// TIA Portal V17 export
// export: Created 2023-02-13T11:16:23.1750279Z, ExportSetting WithDefaults, DisplayName Totally Integrated Automation Portal, DisplayVersion V17, DisplayName TIA Portal Openness, DisplayVersion V17, DisplayName TIA Portal Teamcenter Gateway, DisplayVersion V17, DisplayName TIA Portal Version Control Interface, DisplayVersion V17, DisplayName SINAMICS Startdrive Advanced, DisplayVersion V17, DisplayName SINAMICS Startdrive G130, G150, S120, S150, SINAMICS MV, S210, DisplayVersion V17, DisplayName SINAMICS Startdrive G110M, G120, G120C, G120D, G120P, G115D, DisplayVersion V17, DisplayName STEP 7 Professional, DisplayVersion V17, DisplayName STEP 7 Safety, DisplayVersion V17, DisplayName WinCC Professional, DisplayVersion V17
FUNCTION_BLOCK "IO_Valve_Storage"   // FB1, LAD
{ S7_Optimized_Access := 'FALSE' }
VERSION : 0.1
// stored: AutoNumber true, IsIECCheckEnabled false, SetENOAutomatically false, UDAEnableTagReadback false
   VAR_INPUT
      lock : Bool;
      Init : Bool;
      Reset : Bool;
   END_VAR
   VAR
      "AV-23.01" { S7_SetPoint := 'True'} : "Valve";   // AUTO BUTTERFLY VALVE MAIN INLET PRODUCT TO STORAGE TANK T-23.00
      "AV-23.02" { S7_SetPoint := 'True'} : "Valve";   // AUTO BUTTERFLY VALVE CIP SUPPLY TO STORAGE TANK T-23.00 VIA PIPE INLET
      "AV-23.03" { S7_SetPoint := 'True'} : "Valve";   // AUTO BUTTERFLY VALVE INLET PRODUCT TO STORAGE TANK T-23.00
      "AV-23.04" { S7_SetPoint := 'True'} : "Valve";   // AUTO BUTTERFLY VALVE INLET PRODUCT FROM JBT TO STORAGE TANKS
      "AV-23.05" { S7_SetPoint := 'True'} : "Valve";   // AUTO BUTTERFLY VALVE INLET CIP PRODUCT FROM THE-4 TO STORAGE
      "AV-23.06" { S7_SetPoint := 'True'} : "Valve";   // AUTO BUTTERFLY VALVE OUTLET PRODUCT FROM STORAGE TANK T-23.00
      "AV-23.07" { S7_SetPoint := 'True'} : "Valve";   // AUTO BUTTERFLY VALVE CIP SUPPLY LINE STORAGE TANK T-23.00
      "AV-23.08" { S7_SetPoint := 'True'} : "Valve";   // AUTO BUTTERFLY VALVE CIP SUPPLY STORAGE TANK T-23.00 VIA SPRAY BALL
      "AV-24.01" { S7_SetPoint := 'True'} : "Valve";   // AUTO BUTTERFLY VALVE MAIN INLET PRODUCT TO STORAGE TANK T-24.00
      "AV-24.02" { S7_SetPoint := 'True'} : "Valve";   // AUTO BUTTERFLY VALVE CIP SUPPLY TO STORAGE TANK T-24.00 VIA PIPE INLET
      "AV-24.03" { S7_SetPoint := 'True'} : "Valve";   // AUTO BUTTERFLY VALVE INLET PRODUCT TO STORAGE TANK T-24.00
      "AV-24.04" { S7_SetPoint := 'True'} : "Valve";   // AUTO BUTTERFLY VALVE OUTLET PRODUCT FROM STORAGE TANK T-24.00
      "AV-24.05" { S7_SetPoint := 'True'} : "Valve";   // AUTO BUTTERFLY VALVE CIP SUPPLY LINE STORAGE TANK T-24.00
      "AV-24.06" { S7_SetPoint := 'True'} : "Valve";   // AUTO BUTTERFLY VALVE CIP SUPPLY STORAGE TANK T-24.00 VIA SPRAY BALL
      "AV-24.13" { S7_SetPoint := 'True'} : "Valve";   // AUTO BUTTERFLY VALVE MAIN INLET PRODUCT TO STORAGE TANK T-25.00
      "AV-24.14" { S7_SetPoint := 'True'} : "Valve";   // AUTO BUTTERFLY VALVE CIP SUPPLY TO STORAGE TANK T-25.00 VIA PIPE INLET
      "AV-29.01" { S7_SetPoint := 'True'} : "Valve";   // AUTO BUTTERFLY VALVE INLET PRODUCT TO STORAGE TANK T-25.00
      "AV-29.02" { S7_SetPoint := 'True'} : "Valve";   // AUTO BUTTERFLY VALVE OUTLET PRODUCT FROM STORAGE TANK T-25.00
      "AV-29.03" { S7_SetPoint := 'True'} : "Valve";   // AUTO BUTTERFLY VALVE CIP SUPPLY LINE STORAGE TANK T-25.00
      "AV-29.04" { S7_SetPoint := 'True'} : "Valve";   // AUTO BUTTERFLY VALVE CIP SUPPLY STORAGE TANK T-25.00 VIA SPRAY BALL
      "AV-29.06" { S7_SetPoint := 'True'} : "Valve";   // AUTO BUTTERFLY VALVE CIP SUPPLY STORAGE TANK T-25.00 VIA SPRAY BALL
      "AV-33.01" { S7_SetPoint := 'True'} : "Valve";   // AUTO BUTTERFLY VALVE CIP SUPPLY STORAGE TANKS FROM CIP SUPPLY LINE 3
      "AV-33.02" { S7_SetPoint := 'True'} : "Valve";   // AUTO BUTTERFLY VALVE CIP SUPPLY STORAGE TANK THE-4 JBT FROM CIP SUPPLY LINE 3
      "AV-33.03" { S7_SetPoint := 'True'} : "Valve";   // AUTO BUTTERFLY VALVE CIP SUPPLY STORAGE TANK THE-5 JBT FROM CIP SUPPLY LINE 3
      "AV-33.04" { S7_SetPoint := 'True'} : "Valve";   // AUTO BUTTERFLY VALVE MAIN CIP SUPPLY PRODUCT FROM THE-4 TO STORAGE
      "AV-33.05" { S7_SetPoint := 'True'} : "Valve";   // AUTO BUTTERFLY VALVE MAIN CIP SUPPLY TO STORAGE TANK T-23.00
      "AV-33.06" { S7_SetPoint := 'True'} : "Valve";   // AUTO BUTTERFLY VALVE MAIN CIP SUPPLY LINE STORAGE TANK T-23.00
      "AV-33.07" { S7_SetPoint := 'True'} : "Valve";   // AUTO BUTTERFLY VALVE MAIN CIP SUPPLY TO STORAGE TANK T-24.00
      "AV-33.08" { S7_SetPoint := 'True'} : "Valve";   // AUTO BUTTERFLY VALVE MAIN CIP SUPPLY LINE STORAGE TANK T-24.00
      "AV-33.09" { S7_SetPoint := 'True'} : "Valve";   // AUTO BUTTERFLY VALVE MAIN CIP SUPPLY TO STORAGE TANK T-25.00
      "AV-33.10" { S7_SetPoint := 'True'} : "Valve";
      "AV-33.11" { S7_SetPoint := 'True'} : "Valve";
      "AV-34.01" { S7_SetPoint := 'True'} : "Valve";
      "AV-34.02" { S7_SetPoint := 'True'} : "Valve";
      "AV-34.03" { S7_SetPoint := 'True'} : "Valve";
      "AV-34.04" { S7_SetPoint := 'True'} : "Valve";
      "AV-34.05" { S7_SetPoint := 'True'} : "Valve";
      "AV-34.06" { S7_SetPoint := 'True'} : "Valve";
      "AV-34.07" { S7_SetPoint := 'True'} : "Valve";
      "AV-34.08" { S7_SetPoint := 'True'} : "Valve";
      "AV-34.09" { S7_SetPoint := 'True'} : "Valve";
      "AV-34.10" { S7_SetPoint := 'True'} : "Valve";
      "AV-34.11" { S7_SetPoint := 'True'} : "Valve";
      "AV-34.12" { S7_SetPoint := 'True'} : "Valve";
      "AV-35.01" { S7_SetPoint := 'True'} : "Valve";
      "AV-35.02" { S7_SetPoint := 'True'} : "Valve";
      "AV-35.03" { S7_SetPoint := 'True'} : "Valve";
      "AV-35.04" { S7_SetPoint := 'True'} : "Valve";
      "AV-35.05" { S7_SetPoint := 'True'} : "Valve";
      "AV-35.06" { S7_SetPoint := 'True'} : "Valve";
      "AV-35.07" { S7_SetPoint := 'True'} : "Valve";
      "AV-35.08" { S7_SetPoint := 'True'} : "Valve";
      "AV-39.01" { S7_SetPoint := 'True'} : "Valve";
      "AV-39.02" { S7_SetPoint := 'True'} : "Valve";
      "AV-39.03" { S7_SetPoint := 'True'} : "Valve";
      "AV-39.04" { S7_SetPoint := 'True'} : "Valve";
      "AV-39.06" { S7_SetPoint := 'True'} : "Valve";
      "AV-24.15" { S7_SetPoint := 'True'} : "Valve";
      "AV-24.16" { S7_SetPoint := 'True'} : "Valve";
      "AV-79.01" { S7_SetPoint := 'True'} : "Valve";
      "AV-79.02" { S7_SetPoint := 'True'} : "Valve";
      "AV-79.03" { S7_SetPoint := 'True'} : "Valve";
      "AV-79.04" { S7_SetPoint := 'True'} : "Valve";
      "AV-79.05" { S7_SetPoint := 'True'} : "Valve";
      "AV-79.06" { S7_SetPoint := 'True'} : "Valve";
      "AV-79.07" { S7_SetPoint := 'True'} : "Valve";
      "AV-79.08" { S7_SetPoint := 'True'} : "Valve";
      "AV-79.09" { S7_SetPoint := 'True'} : "Valve";
      "AV-79.10" { S7_SetPoint := 'True'} : "Valve";
      "AV-79.13" { S7_SetPoint := 'True'} : "Valve";
      "AV-79.14" { S7_SetPoint := 'True'} : "Valve";
      "AV-79.15" { S7_SetPoint := 'True'} : "Valve";
      "AV-79.16" { S7_SetPoint := 'True'} : "Valve";
      "AV-79.17" { S7_SetPoint := 'True'} : "Valve";
      "AV-81.01" { S7_SetPoint := 'True'} : "Valve";
      "AV-81.02" { S7_SetPoint := 'True'} : "Valve";
      "AV-81.03" { S7_SetPoint := 'True'} : "Valve";
      "AV-81.04" { S7_SetPoint := 'True'} : "Valve";
      "AV-81.05" { S7_SetPoint := 'True'} : "Valve";
      "AV-81.06" { S7_SetPoint := 'True'} : "Valve";
      "AV-81.07" { S7_SetPoint := 'True'} : "Valve";
      "AV-81.08" { S7_SetPoint := 'True'} : "Valve";
      "AV-81.09" { S7_SetPoint := 'True'} : "Valve";
      "AV-81.10" { S7_SetPoint := 'True'} : "Valve";
      "AV-81.12" { S7_SetPoint := 'True'} : "Valve";
      "AV-81.13" { S7_SetPoint := 'True'} : "Valve";
      "AV-81.14" { S7_SetPoint := 'True'} : "Valve";
      "AV-85.01" { S7_SetPoint := 'True'} : "Valve";
      "AV-85.02" { S7_SetPoint := 'True'} : "Valve";
      "AV-85.03" { S7_SetPoint := 'True'} : "Valve";
      "AV-85.04" { S7_SetPoint := 'True'} : "Valve";
      "AV-85.13" { S7_SetPoint := 'True'} : "Valve";
      "AV-85.12" { S7_SetPoint := 'True'} : "Valve";
      "AV-85.14" { S7_SetPoint := 'True'} : "Valve";
      "AV-85.15" { S7_SetPoint := 'True'} : "Valve";
      "AV-85.05" { S7_SetPoint := 'True'} : "Valve";
      "AV-85.06" { S7_SetPoint := 'True'} : "Valve";
      "AV-85.16" { S7_SetPoint := 'True'} : "Valve";
      "AV-85.17" { S7_SetPoint := 'True'} : "Valve";
      "AV-85.18" { S7_SetPoint := 'True'} : "Valve";
      "AV-85.09" { S7_SetPoint := 'True'} : "Valve";
      "AV-85.08" { S7_SetPoint := 'True'} : "Valve";
      "AV-85.10" { S7_SetPoint := 'True'} : "Valve";
      "AV-85.11" { S7_SetPoint := 'True'} : "Valve";
      "AV-84.05" { S7_SetPoint := 'True'} : "Valve";
      "AV-84.06" { S7_SetPoint := 'True'} : "Valve";
      "AV-84.07" { S7_SetPoint := 'True'} : "Valve";
      "AV-84.08" { S7_SetPoint := 'True'} : "Valve";
      "AV-84.09" { S7_SetPoint := 'True'} : "Valve";
      "AV-84.10" { S7_SetPoint := 'True'} : "Valve";
      "AV-84.12" { S7_SetPoint := 'True'} : "Valve";
      "AV-84.13" { S7_SetPoint := 'True'} : "Valve";
      "AV-84.14" { S7_SetPoint := 'True'} : "Valve";
      "AV-24.09" { S7_SetPoint := 'True'} : "Valve";
      "AV-24.17" { S7_SetPoint := 'True'} : "Valve";
      "AV-24.18" { S7_SetPoint := 'True'} : "Valve";
      "AV-24.19" { S7_SetPoint := 'True'} : "Valve";
      "AV-24.20" { S7_SetPoint := 'True'} : "Valve";
      "AV-24.21" { S7_SetPoint := 'True'} : "Valve";
      "AV-24.22" { S7_SetPoint := 'True'} : "Valve";
      "AV-24.23" { S7_SetPoint := 'True'} : "Valve";
      "AV-24.24" { S7_SetPoint := 'True'} : "Valve";
      "AV-79.21" { S7_SetPoint := 'True'} : "Valve";
      "AV-79.18" { S7_SetPoint := 'True'} : "Valve";
      "AV-79.19" { S7_SetPoint := 'True'} : "Valve";
      "AV-79.20" { S7_SetPoint := 'True'} : "Valve";
   END_VAR
BEGIN

REGION Network 1: AV-23.01
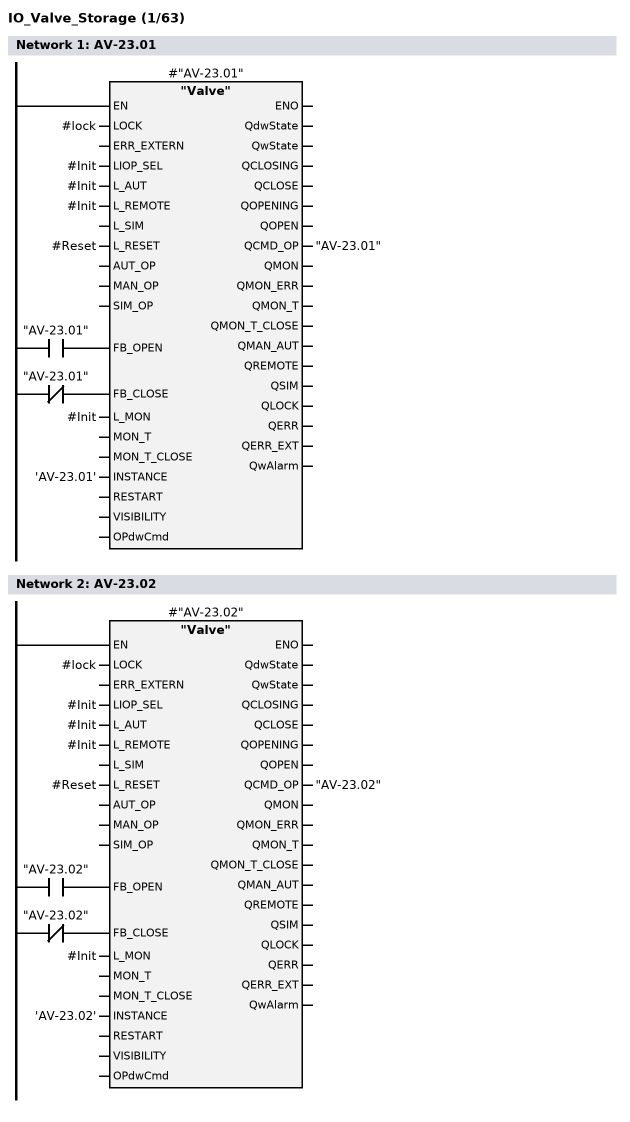
   RUNG wire#powerrail
      #"AV-23.01"(FB_OPEN := wire#w1, FB_CLOSE := wire#w2, LOCK := #lock, ERR_EXTERN :=, LIOP_SEL := #Init, L_AUT := #Init, L_REMOTE := #Init, L_SIM :=, L_RESET := #Reset, AUT_OP :=, MAN_OP :=, SIM_OP :=, L_MON := #Init, MON_T :=, MON_T_CLOSE :=, INSTANCE := 'AV-23.01', RESTART :=, VISIBILITY :=, OPdwCmd :=, QdwState =>, QwState =>, QCLOSING =>, QCLOSE =>, QOPENING =>, QOPEN =>, QCMD_OP => "AV-23.01", QMON =>, QMON_ERR =>, QMON_T =>, QMON_T_CLOSE =>, QMAN_AUT =>, QREMOTE =>, QSIM =>, QLOCK =>, QERR =>, QERR_EXT =>, QwAlarm =>)
   END_RUNG
   RUNG wire#powerrail
      Contact( "AV-23.01" )
   END_RUNG wire#w1
   RUNG wire#powerrail
      I_Contact( "AV-23.01" )
   END_RUNG wire#w2
   // the same network as SCL:
   #"AV-23.01"(LOCK := #lock,   // "Valve"
               LIOP_SEL := #Init,
               L_AUT := #Init,
               L_REMOTE := #Init,
               L_RESET := #Reset,
               FB_OPEN := "AV-23.01",
               FB_CLOSE := NOT "AV-23.01",
               L_MON := #Init,
               INSTANCE := 'AV-23.01',
               QCMD_OP => "AV-23.01");
END_REGION

REGION Network 2: AV-23.02
   RUNG wire#powerrail
      #"AV-23.02"(FB_OPEN := wire#w1, FB_CLOSE := wire#w2, LOCK := #lock, ERR_EXTERN :=, LIOP_SEL := #Init, L_AUT := #Init, L_REMOTE := #Init, L_SIM :=, L_RESET := #Reset, AUT_OP :=, MAN_OP :=, SIM_OP :=, L_MON := #Init, MON_T :=, MON_T_CLOSE :=, INSTANCE := 'AV-23.02', RESTART :=, VISIBILITY :=, OPdwCmd :=, QdwState =>, QwState =>, QCLOSING =>, QCLOSE =>, QOPENING =>, QOPEN =>, QCMD_OP => "AV-23.02", QMON =>, QMON_ERR =>, QMON_T =>, QMON_T_CLOSE =>, QMAN_AUT =>, QREMOTE =>, QSIM =>, QLOCK =>, QERR =>, QERR_EXT =>, QwAlarm =>)
   END_RUNG
   RUNG wire#powerrail
      Contact( "AV-23.02" )
   END_RUNG wire#w1
   RUNG wire#powerrail
      I_Contact( "AV-23.02" )
   END_RUNG wire#w2
   // the same network as SCL:
   #"AV-23.02"(LOCK := #lock,   // "Valve"
               LIOP_SEL := #Init,
               L_AUT := #Init,
               L_REMOTE := #Init,
               L_RESET := #Reset,
               FB_OPEN := "AV-23.02",
               FB_CLOSE := NOT "AV-23.02",
               L_MON := #Init,
               INSTANCE := 'AV-23.02',
               QCMD_OP => "AV-23.02");
END_REGION

REGION Network 3: AV-23.03
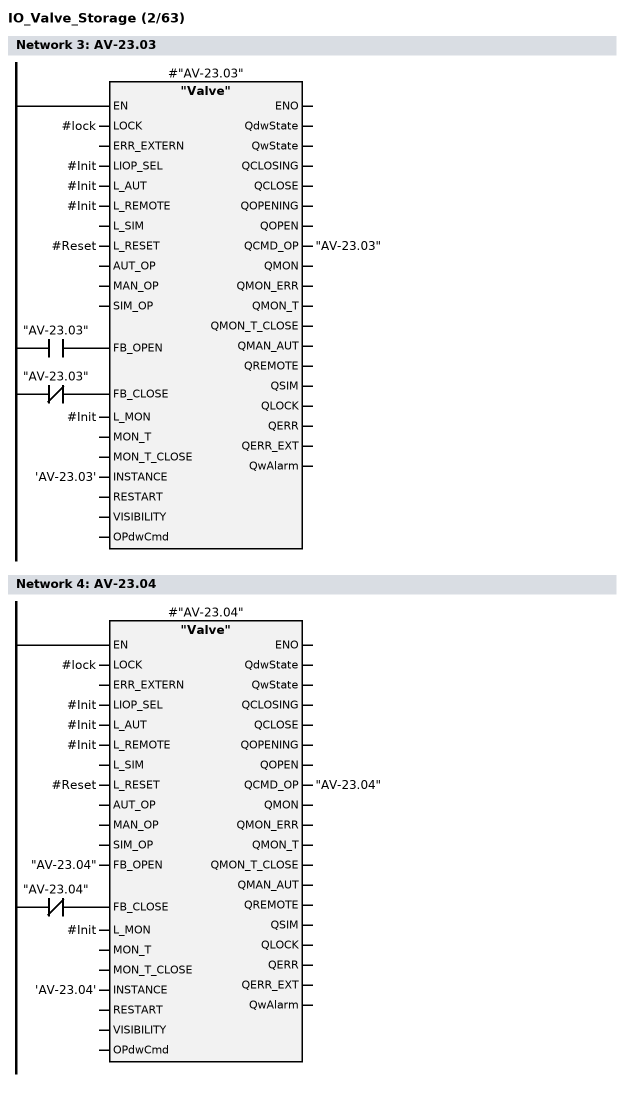
   RUNG wire#powerrail
      #"AV-23.03"(FB_OPEN := wire#w1, FB_CLOSE := wire#w2, LOCK := #lock, ERR_EXTERN :=, LIOP_SEL := #Init, L_AUT := #Init, L_REMOTE := #Init, L_SIM :=, L_RESET := #Reset, AUT_OP :=, MAN_OP :=, SIM_OP :=, L_MON := #Init, MON_T :=, MON_T_CLOSE :=, INSTANCE := 'AV-23.03', RESTART :=, VISIBILITY :=, OPdwCmd :=, QdwState =>, QwState =>, QCLOSING =>, QCLOSE =>, QOPENING =>, QOPEN =>, QCMD_OP => "AV-23.03", QMON =>, QMON_ERR =>, QMON_T =>, QMON_T_CLOSE =>, QMAN_AUT =>, QREMOTE =>, QSIM =>, QLOCK =>, QERR =>, QERR_EXT =>, QwAlarm =>)
   END_RUNG
   RUNG wire#powerrail
      Contact( "AV-23.03" )
   END_RUNG wire#w1
   RUNG wire#powerrail
      I_Contact( "AV-23.03" )
   END_RUNG wire#w2
   // the same network as SCL:
   #"AV-23.03"(LOCK := #lock,   // "Valve"
               LIOP_SEL := #Init,
               L_AUT := #Init,
               L_REMOTE := #Init,
               L_RESET := #Reset,
               FB_OPEN := "AV-23.03",
               FB_CLOSE := NOT "AV-23.03",
               L_MON := #Init,
               INSTANCE := 'AV-23.03',
               QCMD_OP => "AV-23.03");
END_REGION

REGION Network 4: AV-23.04
   RUNG wire#powerrail
      #"AV-23.04"(FB_CLOSE := wire#w1, LOCK := #lock, ERR_EXTERN :=, LIOP_SEL := #Init, L_AUT := #Init, L_REMOTE := #Init, L_SIM :=, L_RESET := #Reset, AUT_OP :=, MAN_OP :=, SIM_OP :=, FB_OPEN := "AV-23.04", L_MON := #Init, MON_T :=, MON_T_CLOSE :=, INSTANCE := 'AV-23.04', RESTART :=, VISIBILITY :=, OPdwCmd :=, QdwState =>, QwState =>, QCLOSING =>, QCLOSE =>, QOPENING =>, QOPEN =>, QCMD_OP => "AV-23.04", QMON =>, QMON_ERR =>, QMON_T =>, QMON_T_CLOSE =>, QMAN_AUT =>, QREMOTE =>, QSIM =>, QLOCK =>, QERR =>, QERR_EXT =>, QwAlarm =>)
   END_RUNG
   RUNG wire#powerrail
      I_Contact( "AV-23.04" )
   END_RUNG wire#w1
   // the same network as SCL:
   #"AV-23.04"(LOCK := #lock,   // "Valve"
               LIOP_SEL := #Init,
               L_AUT := #Init,
               L_REMOTE := #Init,
               L_RESET := #Reset,
               FB_OPEN := "AV-23.04",
               FB_CLOSE := NOT "AV-23.04",
               L_MON := #Init,
               INSTANCE := 'AV-23.04',
               QCMD_OP => "AV-23.04");
END_REGION

REGION Network 5: AV-23.05
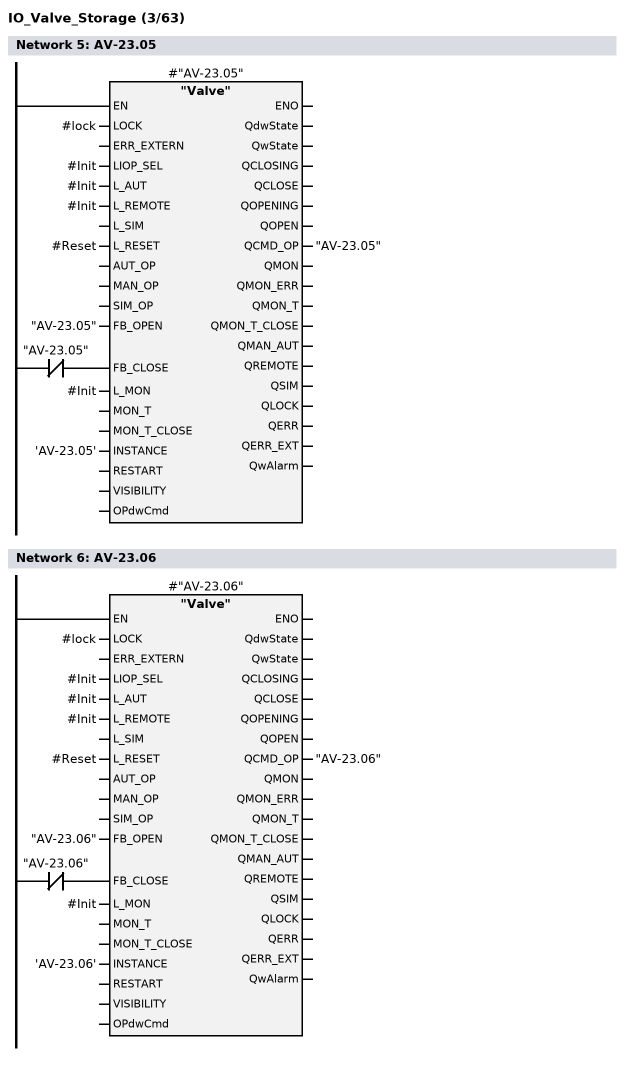
   RUNG wire#powerrail
      #"AV-23.05"(FB_CLOSE := wire#w1, LOCK := #lock, ERR_EXTERN :=, LIOP_SEL := #Init, L_AUT := #Init, L_REMOTE := #Init, L_SIM :=, L_RESET := #Reset, AUT_OP :=, MAN_OP :=, SIM_OP :=, FB_OPEN := "AV-23.05", L_MON := #Init, MON_T :=, MON_T_CLOSE :=, INSTANCE := 'AV-23.05', RESTART :=, VISIBILITY :=, OPdwCmd :=, QdwState =>, QwState =>, QCLOSING =>, QCLOSE =>, QOPENING =>, QOPEN =>, QCMD_OP => "AV-23.05", QMON =>, QMON_ERR =>, QMON_T =>, QMON_T_CLOSE =>, QMAN_AUT =>, QREMOTE =>, QSIM =>, QLOCK =>, QERR =>, QERR_EXT =>, QwAlarm =>)
   END_RUNG
   RUNG wire#powerrail
      I_Contact( "AV-23.05" )
   END_RUNG wire#w1
   // the same network as SCL:
   #"AV-23.05"(LOCK := #lock,   // "Valve"
               LIOP_SEL := #Init,
               L_AUT := #Init,
               L_REMOTE := #Init,
               L_RESET := #Reset,
               FB_OPEN := "AV-23.05",
               FB_CLOSE := NOT "AV-23.05",
               L_MON := #Init,
               INSTANCE := 'AV-23.05',
               QCMD_OP => "AV-23.05");
END_REGION

REGION Network 6: AV-23.06
   RUNG wire#powerrail
      #"AV-23.06"(FB_CLOSE := wire#w1, LOCK := #lock, ERR_EXTERN :=, LIOP_SEL := #Init, L_AUT := #Init, L_REMOTE := #Init, L_SIM :=, L_RESET := #Reset, AUT_OP :=, MAN_OP :=, SIM_OP :=, FB_OPEN := "AV-23.06", L_MON := #Init, MON_T :=, MON_T_CLOSE :=, INSTANCE := 'AV-23.06', RESTART :=, VISIBILITY :=, OPdwCmd :=, QdwState =>, QwState =>, QCLOSING =>, QCLOSE =>, QOPENING =>, QOPEN =>, QCMD_OP => "AV-23.06", QMON =>, QMON_ERR =>, QMON_T =>, QMON_T_CLOSE =>, QMAN_AUT =>, QREMOTE =>, QSIM =>, QLOCK =>, QERR =>, QERR_EXT =>, QwAlarm =>)
   END_RUNG
   RUNG wire#powerrail
      I_Contact( "AV-23.06" )
   END_RUNG wire#w1
   // the same network as SCL:
   #"AV-23.06"(LOCK := #lock,   // "Valve"
               LIOP_SEL := #Init,
               L_AUT := #Init,
               L_REMOTE := #Init,
               L_RESET := #Reset,
               FB_OPEN := "AV-23.06",
               FB_CLOSE := NOT "AV-23.06",
               L_MON := #Init,
               INSTANCE := 'AV-23.06',
               QCMD_OP => "AV-23.06");
END_REGION

REGION Network 7: AV-23.07
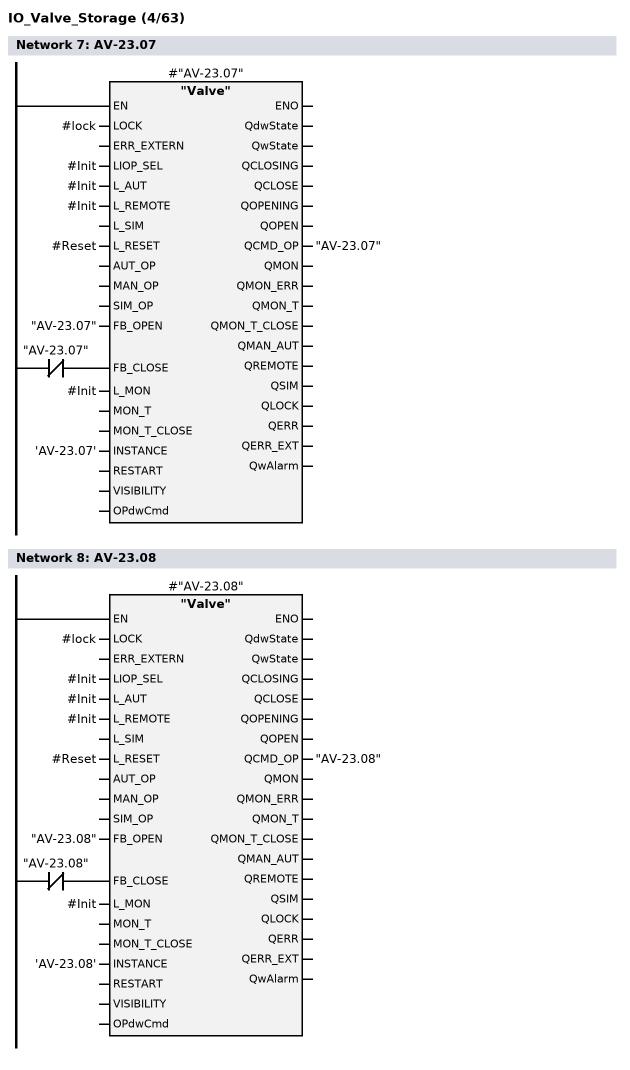
   RUNG wire#powerrail
      #"AV-23.07"(FB_CLOSE := wire#w1, LOCK := #lock, ERR_EXTERN :=, LIOP_SEL := #Init, L_AUT := #Init, L_REMOTE := #Init, L_SIM :=, L_RESET := #Reset, AUT_OP :=, MAN_OP :=, SIM_OP :=, FB_OPEN := "AV-23.07", L_MON := #Init, MON_T :=, MON_T_CLOSE :=, INSTANCE := 'AV-23.07', RESTART :=, VISIBILITY :=, OPdwCmd :=, QdwState =>, QwState =>, QCLOSING =>, QCLOSE =>, QOPENING =>, QOPEN =>, QCMD_OP => "AV-23.07", QMON =>, QMON_ERR =>, QMON_T =>, QMON_T_CLOSE =>, QMAN_AUT =>, QREMOTE =>, QSIM =>, QLOCK =>, QERR =>, QERR_EXT =>, QwAlarm =>)
   END_RUNG
   RUNG wire#powerrail
      I_Contact( "AV-23.07" )
   END_RUNG wire#w1
   // the same network as SCL:
   #"AV-23.07"(LOCK := #lock,   // "Valve"
               LIOP_SEL := #Init,
               L_AUT := #Init,
               L_REMOTE := #Init,
               L_RESET := #Reset,
               FB_OPEN := "AV-23.07",
               FB_CLOSE := NOT "AV-23.07",
               L_MON := #Init,
               INSTANCE := 'AV-23.07',
               QCMD_OP => "AV-23.07");
END_REGION

REGION Network 8: AV-23.08
   RUNG wire#powerrail
      #"AV-23.08"(FB_CLOSE := wire#w1, LOCK := #lock, ERR_EXTERN :=, LIOP_SEL := #Init, L_AUT := #Init, L_REMOTE := #Init, L_SIM :=, L_RESET := #Reset, AUT_OP :=, MAN_OP :=, SIM_OP :=, FB_OPEN := "AV-23.08", L_MON := #Init, MON_T :=, MON_T_CLOSE :=, INSTANCE := 'AV-23.08', RESTART :=, VISIBILITY :=, OPdwCmd :=, QdwState =>, QwState =>, QCLOSING =>, QCLOSE =>, QOPENING =>, QOPEN =>, QCMD_OP => "AV-23.08", QMON =>, QMON_ERR =>, QMON_T =>, QMON_T_CLOSE =>, QMAN_AUT =>, QREMOTE =>, QSIM =>, QLOCK =>, QERR =>, QERR_EXT =>, QwAlarm =>)
   END_RUNG
   RUNG wire#powerrail
      I_Contact( "AV-23.08" )
   END_RUNG wire#w1
   // the same network as SCL:
   #"AV-23.08"(LOCK := #lock,   // "Valve"
               LIOP_SEL := #Init,
               L_AUT := #Init,
               L_REMOTE := #Init,
               L_RESET := #Reset,
               FB_OPEN := "AV-23.08",
               FB_CLOSE := NOT "AV-23.08",
               L_MON := #Init,
               INSTANCE := 'AV-23.08',
               QCMD_OP => "AV-23.08");
END_REGION

REGION Network 10: AV-24.01
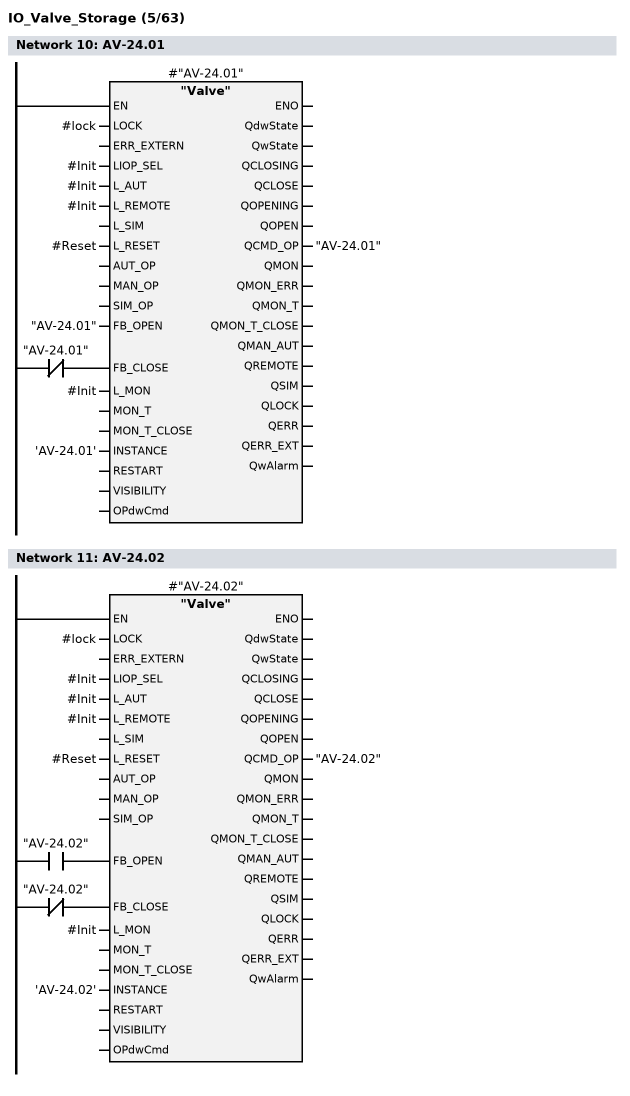
   RUNG wire#powerrail
      #"AV-24.01"(FB_CLOSE := wire#w1, LOCK := #lock, ERR_EXTERN :=, LIOP_SEL := #Init, L_AUT := #Init, L_REMOTE := #Init, L_SIM :=, L_RESET := #Reset, AUT_OP :=, MAN_OP :=, SIM_OP :=, FB_OPEN := "AV-24.01", L_MON := #Init, MON_T :=, MON_T_CLOSE :=, INSTANCE := 'AV-24.01', RESTART :=, VISIBILITY :=, OPdwCmd :=, QdwState =>, QwState =>, QCLOSING =>, QCLOSE =>, QOPENING =>, QOPEN =>, QCMD_OP => "AV-24.01", QMON =>, QMON_ERR =>, QMON_T =>, QMON_T_CLOSE =>, QMAN_AUT =>, QREMOTE =>, QSIM =>, QLOCK =>, QERR =>, QERR_EXT =>, QwAlarm =>)
   END_RUNG
   RUNG wire#powerrail
      I_Contact( "AV-24.01" )
   END_RUNG wire#w1
   // the same network as SCL:
   #"AV-24.01"(LOCK := #lock,   // "Valve"
               LIOP_SEL := #Init,
               L_AUT := #Init,
               L_REMOTE := #Init,
               L_RESET := #Reset,
               FB_OPEN := "AV-24.01",
               FB_CLOSE := NOT "AV-24.01",
               L_MON := #Init,
               INSTANCE := 'AV-24.01',
               QCMD_OP => "AV-24.01");
END_REGION

REGION Network 11: AV-24.02
   RUNG wire#powerrail
      #"AV-24.02"(FB_OPEN := wire#w1, FB_CLOSE := wire#w2, LOCK := #lock, ERR_EXTERN :=, LIOP_SEL := #Init, L_AUT := #Init, L_REMOTE := #Init, L_SIM :=, L_RESET := #Reset, AUT_OP :=, MAN_OP :=, SIM_OP :=, L_MON := #Init, MON_T :=, MON_T_CLOSE :=, INSTANCE := 'AV-24.02', RESTART :=, VISIBILITY :=, OPdwCmd :=, QdwState =>, QwState =>, QCLOSING =>, QCLOSE =>, QOPENING =>, QOPEN =>, QCMD_OP => "AV-24.02", QMON =>, QMON_ERR =>, QMON_T =>, QMON_T_CLOSE =>, QMAN_AUT =>, QREMOTE =>, QSIM =>, QLOCK =>, QERR =>, QERR_EXT =>, QwAlarm =>)
   END_RUNG
   RUNG wire#powerrail
      Contact( "AV-24.02" )
   END_RUNG wire#w1
   RUNG wire#powerrail
      I_Contact( "AV-24.02" )
   END_RUNG wire#w2
   // the same network as SCL:
   #"AV-24.02"(LOCK := #lock,   // "Valve"
               LIOP_SEL := #Init,
               L_AUT := #Init,
               L_REMOTE := #Init,
               L_RESET := #Reset,
               FB_OPEN := "AV-24.02",
               FB_CLOSE := NOT "AV-24.02",
               L_MON := #Init,
               INSTANCE := 'AV-24.02',
               QCMD_OP => "AV-24.02");
END_REGION

REGION Network 12: AV-24.03
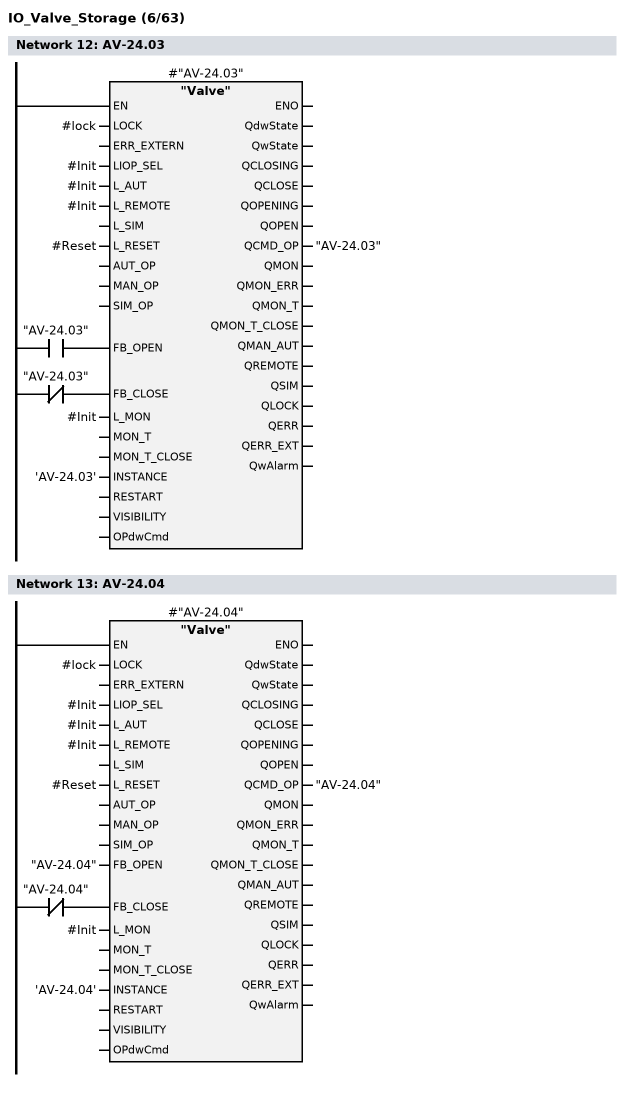
   RUNG wire#powerrail
      #"AV-24.03"(FB_OPEN := wire#w1, FB_CLOSE := wire#w2, LOCK := #lock, ERR_EXTERN :=, LIOP_SEL := #Init, L_AUT := #Init, L_REMOTE := #Init, L_SIM :=, L_RESET := #Reset, AUT_OP :=, MAN_OP :=, SIM_OP :=, L_MON := #Init, MON_T :=, MON_T_CLOSE :=, INSTANCE := 'AV-24.03', RESTART :=, VISIBILITY :=, OPdwCmd :=, QdwState =>, QwState =>, QCLOSING =>, QCLOSE =>, QOPENING =>, QOPEN =>, QCMD_OP => "AV-24.03", QMON =>, QMON_ERR =>, QMON_T =>, QMON_T_CLOSE =>, QMAN_AUT =>, QREMOTE =>, QSIM =>, QLOCK =>, QERR =>, QERR_EXT =>, QwAlarm =>)
   END_RUNG
   RUNG wire#powerrail
      Contact( "AV-24.03" )
   END_RUNG wire#w1
   RUNG wire#powerrail
      I_Contact( "AV-24.03" )
   END_RUNG wire#w2
   // the same network as SCL:
   #"AV-24.03"(LOCK := #lock,   // "Valve"
               LIOP_SEL := #Init,
               L_AUT := #Init,
               L_REMOTE := #Init,
               L_RESET := #Reset,
               FB_OPEN := "AV-24.03",
               FB_CLOSE := NOT "AV-24.03",
               L_MON := #Init,
               INSTANCE := 'AV-24.03',
               QCMD_OP => "AV-24.03");
END_REGION

REGION Network 13: AV-24.04
   RUNG wire#powerrail
      #"AV-24.04"(FB_CLOSE := wire#w1, LOCK := #lock, ERR_EXTERN :=, LIOP_SEL := #Init, L_AUT := #Init, L_REMOTE := #Init, L_SIM :=, L_RESET := #Reset, AUT_OP :=, MAN_OP :=, SIM_OP :=, FB_OPEN := "AV-24.04", L_MON := #Init, MON_T :=, MON_T_CLOSE :=, INSTANCE := 'AV-24.04', RESTART :=, VISIBILITY :=, OPdwCmd :=, QdwState =>, QwState =>, QCLOSING =>, QCLOSE =>, QOPENING =>, QOPEN =>, QCMD_OP => "AV-24.04", QMON =>, QMON_ERR =>, QMON_T =>, QMON_T_CLOSE =>, QMAN_AUT =>, QREMOTE =>, QSIM =>, QLOCK =>, QERR =>, QERR_EXT =>, QwAlarm =>)
   END_RUNG
   RUNG wire#powerrail
      I_Contact( "AV-24.04" )
   END_RUNG wire#w1
   // the same network as SCL:
   #"AV-24.04"(LOCK := #lock,   // "Valve"
               LIOP_SEL := #Init,
               L_AUT := #Init,
               L_REMOTE := #Init,
               L_RESET := #Reset,
               FB_OPEN := "AV-24.04",
               FB_CLOSE := NOT "AV-24.04",
               L_MON := #Init,
               INSTANCE := 'AV-24.04',
               QCMD_OP => "AV-24.04");
END_REGION

REGION Network 14: AV-24.05
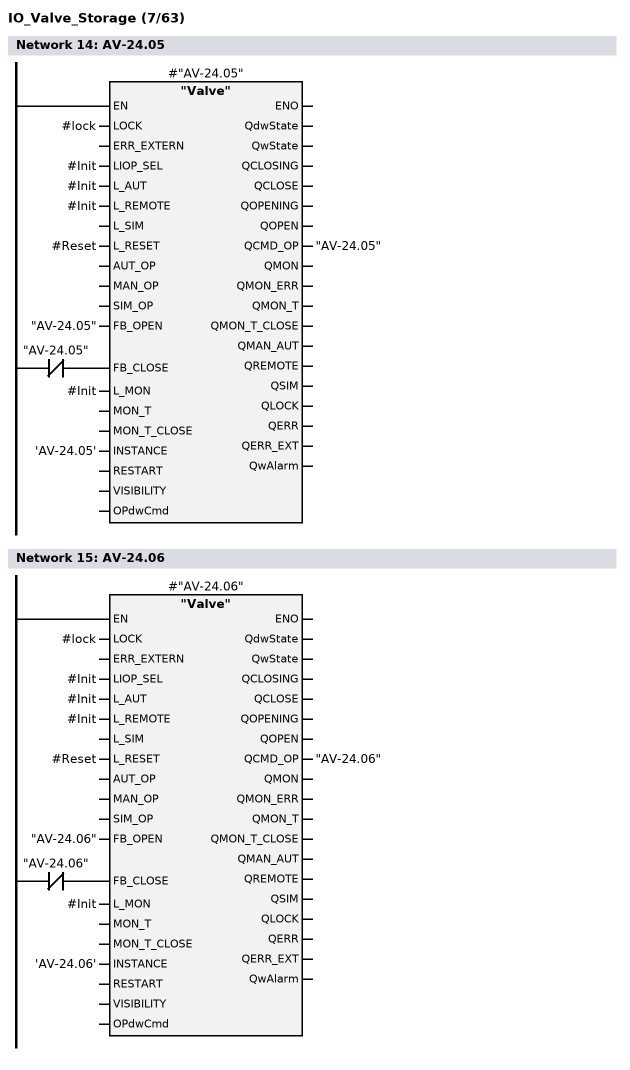
   RUNG wire#powerrail
      #"AV-24.05"(FB_CLOSE := wire#w1, LOCK := #lock, ERR_EXTERN :=, LIOP_SEL := #Init, L_AUT := #Init, L_REMOTE := #Init, L_SIM :=, L_RESET := #Reset, AUT_OP :=, MAN_OP :=, SIM_OP :=, FB_OPEN := "AV-24.05", L_MON := #Init, MON_T :=, MON_T_CLOSE :=, INSTANCE := 'AV-24.05', RESTART :=, VISIBILITY :=, OPdwCmd :=, QdwState =>, QwState =>, QCLOSING =>, QCLOSE =>, QOPENING =>, QOPEN =>, QCMD_OP => "AV-24.05", QMON =>, QMON_ERR =>, QMON_T =>, QMON_T_CLOSE =>, QMAN_AUT =>, QREMOTE =>, QSIM =>, QLOCK =>, QERR =>, QERR_EXT =>, QwAlarm =>)
   END_RUNG
   RUNG wire#powerrail
      I_Contact( "AV-24.05" )
   END_RUNG wire#w1
   // the same network as SCL:
   #"AV-24.05"(LOCK := #lock,   // "Valve"
               LIOP_SEL := #Init,
               L_AUT := #Init,
               L_REMOTE := #Init,
               L_RESET := #Reset,
               FB_OPEN := "AV-24.05",
               FB_CLOSE := NOT "AV-24.05",
               L_MON := #Init,
               INSTANCE := 'AV-24.05',
               QCMD_OP => "AV-24.05");
END_REGION

REGION Network 15: AV-24.06
   RUNG wire#powerrail
      #"AV-24.06"(FB_CLOSE := wire#w1, LOCK := #lock, ERR_EXTERN :=, LIOP_SEL := #Init, L_AUT := #Init, L_REMOTE := #Init, L_SIM :=, L_RESET := #Reset, AUT_OP :=, MAN_OP :=, SIM_OP :=, FB_OPEN := "AV-24.06", L_MON := #Init, MON_T :=, MON_T_CLOSE :=, INSTANCE := 'AV-24.06', RESTART :=, VISIBILITY :=, OPdwCmd :=, QdwState =>, QwState =>, QCLOSING =>, QCLOSE =>, QOPENING =>, QOPEN =>, QCMD_OP => "AV-24.06", QMON =>, QMON_ERR =>, QMON_T =>, QMON_T_CLOSE =>, QMAN_AUT =>, QREMOTE =>, QSIM =>, QLOCK =>, QERR =>, QERR_EXT =>, QwAlarm =>)
   END_RUNG
   RUNG wire#powerrail
      I_Contact( "AV-24.06" )
   END_RUNG wire#w1
   // the same network as SCL:
   #"AV-24.06"(LOCK := #lock,   // "Valve"
               LIOP_SEL := #Init,
               L_AUT := #Init,
               L_REMOTE := #Init,
               L_RESET := #Reset,
               FB_OPEN := "AV-24.06",
               FB_CLOSE := NOT "AV-24.06",
               L_MON := #Init,
               INSTANCE := 'AV-24.06',
               QCMD_OP => "AV-24.06");
END_REGION

REGION Network 16: AV-24.09
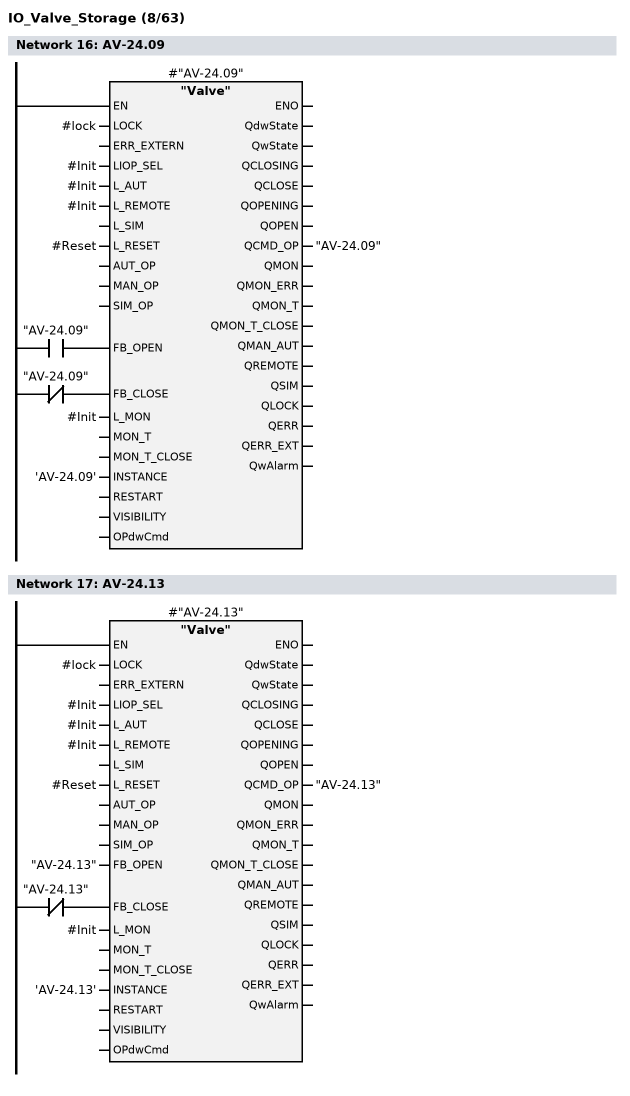
   RUNG wire#powerrail
      #"AV-24.09"(FB_OPEN := wire#w1, FB_CLOSE := wire#w2, LOCK := #lock, ERR_EXTERN :=, LIOP_SEL := #Init, L_AUT := #Init, L_REMOTE := #Init, L_SIM :=, L_RESET := #Reset, AUT_OP :=, MAN_OP :=, SIM_OP :=, L_MON := #Init, MON_T :=, MON_T_CLOSE :=, INSTANCE := 'AV-24.09', RESTART :=, VISIBILITY :=, OPdwCmd :=, QdwState =>, QwState =>, QCLOSING =>, QCLOSE =>, QOPENING =>, QOPEN =>, QCMD_OP => "AV-24.09", QMON =>, QMON_ERR =>, QMON_T =>, QMON_T_CLOSE =>, QMAN_AUT =>, QREMOTE =>, QSIM =>, QLOCK =>, QERR =>, QERR_EXT =>, QwAlarm =>)
   END_RUNG
   RUNG wire#powerrail
      Contact( "AV-24.09" )
   END_RUNG wire#w1
   RUNG wire#powerrail
      I_Contact( "AV-24.09" )
   END_RUNG wire#w2
   // the same network as SCL:
   #"AV-24.09"(LOCK := #lock,   // "Valve"
               LIOP_SEL := #Init,
               L_AUT := #Init,
               L_REMOTE := #Init,
               L_RESET := #Reset,
               FB_OPEN := "AV-24.09",
               FB_CLOSE := NOT "AV-24.09",
               L_MON := #Init,
               INSTANCE := 'AV-24.09',
               QCMD_OP => "AV-24.09");
END_REGION

REGION Network 17: AV-24.13
   RUNG wire#powerrail
      #"AV-24.13"(FB_CLOSE := wire#w1, LOCK := #lock, ERR_EXTERN :=, LIOP_SEL := #Init, L_AUT := #Init, L_REMOTE := #Init, L_SIM :=, L_RESET := #Reset, AUT_OP :=, MAN_OP :=, SIM_OP :=, FB_OPEN := "AV-24.13", L_MON := #Init, MON_T :=, MON_T_CLOSE :=, INSTANCE := 'AV-24.13', RESTART :=, VISIBILITY :=, OPdwCmd :=, QdwState =>, QwState =>, QCLOSING =>, QCLOSE =>, QOPENING =>, QOPEN =>, QCMD_OP => "AV-24.13", QMON =>, QMON_ERR =>, QMON_T =>, QMON_T_CLOSE =>, QMAN_AUT =>, QREMOTE =>, QSIM =>, QLOCK =>, QERR =>, QERR_EXT =>, QwAlarm =>)
   END_RUNG
   RUNG wire#powerrail
      I_Contact( "AV-24.13" )
   END_RUNG wire#w1
   // the same network as SCL:
   #"AV-24.13"(LOCK := #lock,   // "Valve"
               LIOP_SEL := #Init,
               L_AUT := #Init,
               L_REMOTE := #Init,
               L_RESET := #Reset,
               FB_OPEN := "AV-24.13",
               FB_CLOSE := NOT "AV-24.13",
               L_MON := #Init,
               INSTANCE := 'AV-24.13',
               QCMD_OP => "AV-24.13");
END_REGION

REGION Network 18: AV-24.14
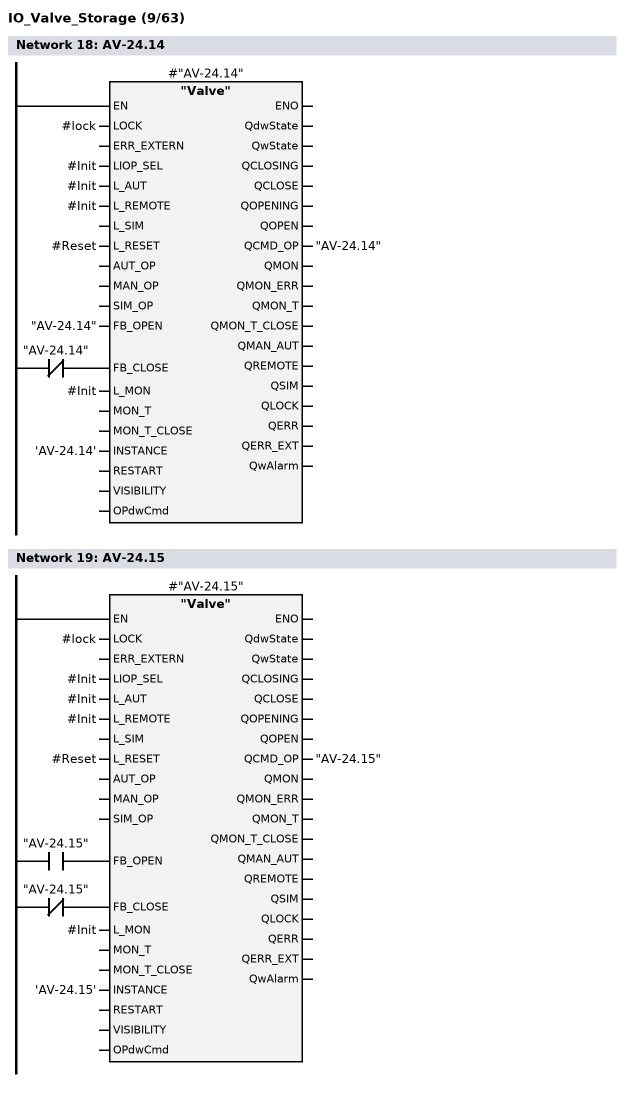
   RUNG wire#powerrail
      #"AV-24.14"(FB_CLOSE := wire#w1, LOCK := #lock, ERR_EXTERN :=, LIOP_SEL := #Init, L_AUT := #Init, L_REMOTE := #Init, L_SIM :=, L_RESET := #Reset, AUT_OP :=, MAN_OP :=, SIM_OP :=, FB_OPEN := "AV-24.14", L_MON := #Init, MON_T :=, MON_T_CLOSE :=, INSTANCE := 'AV-24.14', RESTART :=, VISIBILITY :=, OPdwCmd :=, QdwState =>, QwState =>, QCLOSING =>, QCLOSE =>, QOPENING =>, QOPEN =>, QCMD_OP => "AV-24.14", QMON =>, QMON_ERR =>, QMON_T =>, QMON_T_CLOSE =>, QMAN_AUT =>, QREMOTE =>, QSIM =>, QLOCK =>, QERR =>, QERR_EXT =>, QwAlarm =>)
   END_RUNG
   RUNG wire#powerrail
      I_Contact( "AV-24.14" )
   END_RUNG wire#w1
   // the same network as SCL:
   #"AV-24.14"(LOCK := #lock,   // "Valve"
               LIOP_SEL := #Init,
               L_AUT := #Init,
               L_REMOTE := #Init,
               L_RESET := #Reset,
               FB_OPEN := "AV-24.14",
               FB_CLOSE := NOT "AV-24.14",
               L_MON := #Init,
               INSTANCE := 'AV-24.14',
               QCMD_OP => "AV-24.14");
END_REGION

REGION Network 19: AV-24.15
   RUNG wire#powerrail
      #"AV-24.15"(FB_OPEN := wire#w1, FB_CLOSE := wire#w2, LOCK := #lock, ERR_EXTERN :=, LIOP_SEL := #Init, L_AUT := #Init, L_REMOTE := #Init, L_SIM :=, L_RESET := #Reset, AUT_OP :=, MAN_OP :=, SIM_OP :=, L_MON := #Init, MON_T :=, MON_T_CLOSE :=, INSTANCE := 'AV-24.15', RESTART :=, VISIBILITY :=, OPdwCmd :=, QdwState =>, QwState =>, QCLOSING =>, QCLOSE =>, QOPENING =>, QOPEN =>, QCMD_OP => "AV-24.15", QMON =>, QMON_ERR =>, QMON_T =>, QMON_T_CLOSE =>, QMAN_AUT =>, QREMOTE =>, QSIM =>, QLOCK =>, QERR =>, QERR_EXT =>, QwAlarm =>)
   END_RUNG
   RUNG wire#powerrail
      Contact( "AV-24.15" )
   END_RUNG wire#w1
   RUNG wire#powerrail
      I_Contact( "AV-24.15" )
   END_RUNG wire#w2
   // the same network as SCL:
   #"AV-24.15"(LOCK := #lock,   // "Valve"
               LIOP_SEL := #Init,
               L_AUT := #Init,
               L_REMOTE := #Init,
               L_RESET := #Reset,
               FB_OPEN := "AV-24.15",
               FB_CLOSE := NOT "AV-24.15",
               L_MON := #Init,
               INSTANCE := 'AV-24.15',
               QCMD_OP => "AV-24.15");
END_REGION

REGION Network 20: AV-24.16
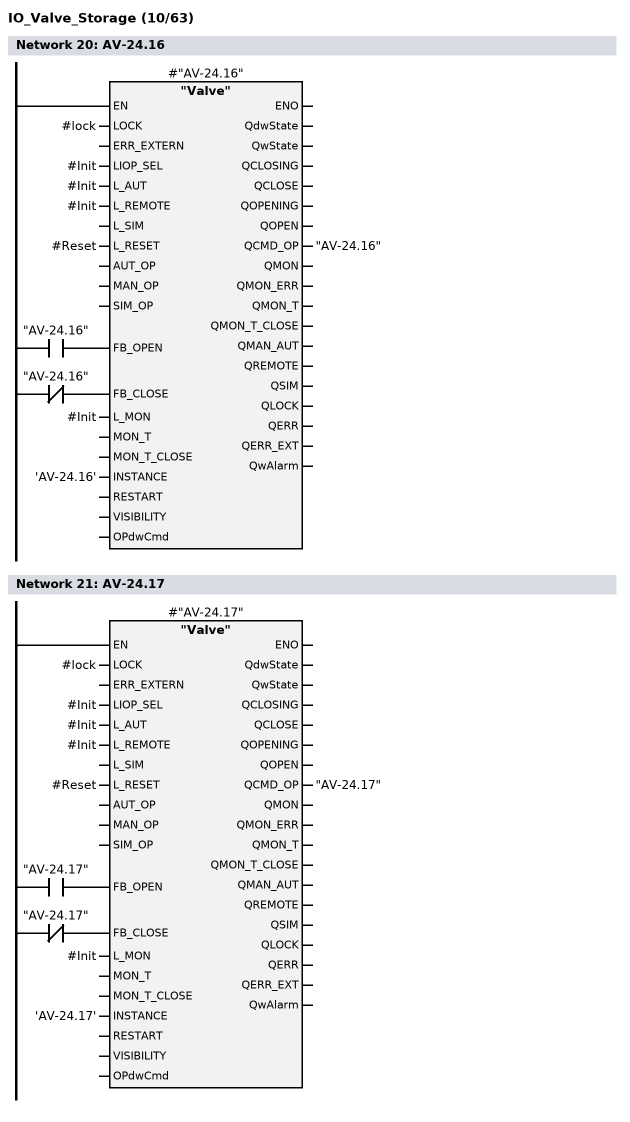
   RUNG wire#powerrail
      #"AV-24.16"(FB_OPEN := wire#w1, FB_CLOSE := wire#w2, LOCK := #lock, ERR_EXTERN :=, LIOP_SEL := #Init, L_AUT := #Init, L_REMOTE := #Init, L_SIM :=, L_RESET := #Reset, AUT_OP :=, MAN_OP :=, SIM_OP :=, L_MON := #Init, MON_T :=, MON_T_CLOSE :=, INSTANCE := 'AV-24.16', RESTART :=, VISIBILITY :=, OPdwCmd :=, QdwState =>, QwState =>, QCLOSING =>, QCLOSE =>, QOPENING =>, QOPEN =>, QCMD_OP => "AV-24.16", QMON =>, QMON_ERR =>, QMON_T =>, QMON_T_CLOSE =>, QMAN_AUT =>, QREMOTE =>, QSIM =>, QLOCK =>, QERR =>, QERR_EXT =>, QwAlarm =>)
   END_RUNG
   RUNG wire#powerrail
      Contact( "AV-24.16" )
   END_RUNG wire#w1
   RUNG wire#powerrail
      I_Contact( "AV-24.16" )
   END_RUNG wire#w2
   // the same network as SCL:
   #"AV-24.16"(LOCK := #lock,   // "Valve"
               LIOP_SEL := #Init,
               L_AUT := #Init,
               L_REMOTE := #Init,
               L_RESET := #Reset,
               FB_OPEN := "AV-24.16",
               FB_CLOSE := NOT "AV-24.16",
               L_MON := #Init,
               INSTANCE := 'AV-24.16',
               QCMD_OP => "AV-24.16");
END_REGION

REGION Network 21: AV-24.17
   RUNG wire#powerrail
      #"AV-24.17"(FB_OPEN := wire#w1, FB_CLOSE := wire#w2, LOCK := #lock, ERR_EXTERN :=, LIOP_SEL := #Init, L_AUT := #Init, L_REMOTE := #Init, L_SIM :=, L_RESET := #Reset, AUT_OP :=, MAN_OP :=, SIM_OP :=, L_MON := #Init, MON_T :=, MON_T_CLOSE :=, INSTANCE := 'AV-24.17', RESTART :=, VISIBILITY :=, OPdwCmd :=, QdwState =>, QwState =>, QCLOSING =>, QCLOSE =>, QOPENING =>, QOPEN =>, QCMD_OP => "AV-24.17", QMON =>, QMON_ERR =>, QMON_T =>, QMON_T_CLOSE =>, QMAN_AUT =>, QREMOTE =>, QSIM =>, QLOCK =>, QERR =>, QERR_EXT =>, QwAlarm =>)
   END_RUNG
   RUNG wire#powerrail
      Contact( "AV-24.17" )
   END_RUNG wire#w1
   RUNG wire#powerrail
      I_Contact( "AV-24.17" )
   END_RUNG wire#w2
   // the same network as SCL:
   #"AV-24.17"(LOCK := #lock,   // "Valve"
               LIOP_SEL := #Init,
               L_AUT := #Init,
               L_REMOTE := #Init,
               L_RESET := #Reset,
               FB_OPEN := "AV-24.17",
               FB_CLOSE := NOT "AV-24.17",
               L_MON := #Init,
               INSTANCE := 'AV-24.17',
               QCMD_OP => "AV-24.17");
END_REGION

REGION Network 22: AV-24.18
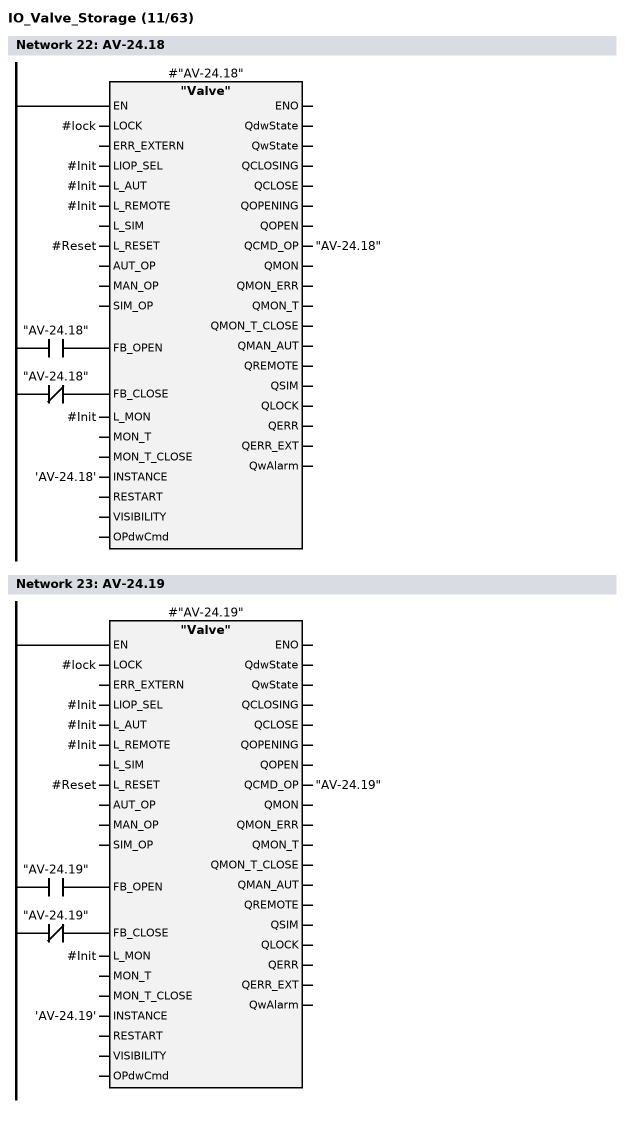
   RUNG wire#powerrail
      #"AV-24.18"(FB_OPEN := wire#w1, FB_CLOSE := wire#w2, LOCK := #lock, ERR_EXTERN :=, LIOP_SEL := #Init, L_AUT := #Init, L_REMOTE := #Init, L_SIM :=, L_RESET := #Reset, AUT_OP :=, MAN_OP :=, SIM_OP :=, L_MON := #Init, MON_T :=, MON_T_CLOSE :=, INSTANCE := 'AV-24.18', RESTART :=, VISIBILITY :=, OPdwCmd :=, QdwState =>, QwState =>, QCLOSING =>, QCLOSE =>, QOPENING =>, QOPEN =>, QCMD_OP => "AV-24.18", QMON =>, QMON_ERR =>, QMON_T =>, QMON_T_CLOSE =>, QMAN_AUT =>, QREMOTE =>, QSIM =>, QLOCK =>, QERR =>, QERR_EXT =>, QwAlarm =>)
   END_RUNG
   RUNG wire#powerrail
      Contact( "AV-24.18" )
   END_RUNG wire#w1
   RUNG wire#powerrail
      I_Contact( "AV-24.18" )
   END_RUNG wire#w2
   // the same network as SCL:
   #"AV-24.18"(LOCK := #lock,   // "Valve"
               LIOP_SEL := #Init,
               L_AUT := #Init,
               L_REMOTE := #Init,
               L_RESET := #Reset,
               FB_OPEN := "AV-24.18",
               FB_CLOSE := NOT "AV-24.18",
               L_MON := #Init,
               INSTANCE := 'AV-24.18',
               QCMD_OP => "AV-24.18");
END_REGION

REGION Network 23: AV-24.19
   RUNG wire#powerrail
      #"AV-24.19"(FB_OPEN := wire#w1, FB_CLOSE := wire#w2, LOCK := #lock, ERR_EXTERN :=, LIOP_SEL := #Init, L_AUT := #Init, L_REMOTE := #Init, L_SIM :=, L_RESET := #Reset, AUT_OP :=, MAN_OP :=, SIM_OP :=, L_MON := #Init, MON_T :=, MON_T_CLOSE :=, INSTANCE := 'AV-24.19', RESTART :=, VISIBILITY :=, OPdwCmd :=, QdwState =>, QwState =>, QCLOSING =>, QCLOSE =>, QOPENING =>, QOPEN =>, QCMD_OP => "AV-24.19", QMON =>, QMON_ERR =>, QMON_T =>, QMON_T_CLOSE =>, QMAN_AUT =>, QREMOTE =>, QSIM =>, QLOCK =>, QERR =>, QERR_EXT =>, QwAlarm =>)
   END_RUNG
   RUNG wire#powerrail
      Contact( "AV-24.19" )
   END_RUNG wire#w1
   RUNG wire#powerrail
      I_Contact( "AV-24.19" )
   END_RUNG wire#w2
   // the same network as SCL:
   #"AV-24.19"(LOCK := #lock,   // "Valve"
               LIOP_SEL := #Init,
               L_AUT := #Init,
               L_REMOTE := #Init,
               L_RESET := #Reset,
               FB_OPEN := "AV-24.19",
               FB_CLOSE := NOT "AV-24.19",
               L_MON := #Init,
               INSTANCE := 'AV-24.19',
               QCMD_OP => "AV-24.19");
END_REGION

REGION Network 24: AV-24.20
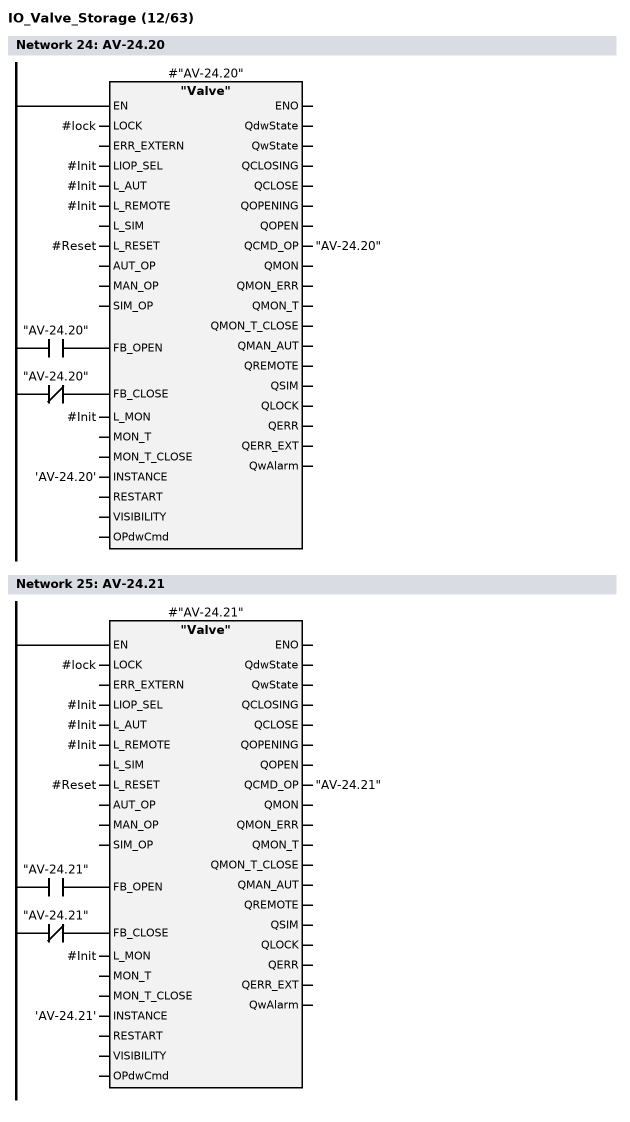
   RUNG wire#powerrail
      #"AV-24.20"(FB_OPEN := wire#w1, FB_CLOSE := wire#w2, LOCK := #lock, ERR_EXTERN :=, LIOP_SEL := #Init, L_AUT := #Init, L_REMOTE := #Init, L_SIM :=, L_RESET := #Reset, AUT_OP :=, MAN_OP :=, SIM_OP :=, L_MON := #Init, MON_T :=, MON_T_CLOSE :=, INSTANCE := 'AV-24.20', RESTART :=, VISIBILITY :=, OPdwCmd :=, QdwState =>, QwState =>, QCLOSING =>, QCLOSE =>, QOPENING =>, QOPEN =>, QCMD_OP => "AV-24.20", QMON =>, QMON_ERR =>, QMON_T =>, QMON_T_CLOSE =>, QMAN_AUT =>, QREMOTE =>, QSIM =>, QLOCK =>, QERR =>, QERR_EXT =>, QwAlarm =>)
   END_RUNG
   RUNG wire#powerrail
      Contact( "AV-24.20" )
   END_RUNG wire#w1
   RUNG wire#powerrail
      I_Contact( "AV-24.20" )
   END_RUNG wire#w2
   // the same network as SCL:
   #"AV-24.20"(LOCK := #lock,   // "Valve"
               LIOP_SEL := #Init,
               L_AUT := #Init,
               L_REMOTE := #Init,
               L_RESET := #Reset,
               FB_OPEN := "AV-24.20",
               FB_CLOSE := NOT "AV-24.20",
               L_MON := #Init,
               INSTANCE := 'AV-24.20',
               QCMD_OP => "AV-24.20");
END_REGION

REGION Network 25: AV-24.21
   RUNG wire#powerrail
      #"AV-24.21"(FB_OPEN := wire#w1, FB_CLOSE := wire#w2, LOCK := #lock, ERR_EXTERN :=, LIOP_SEL := #Init, L_AUT := #Init, L_REMOTE := #Init, L_SIM :=, L_RESET := #Reset, AUT_OP :=, MAN_OP :=, SIM_OP :=, L_MON := #Init, MON_T :=, MON_T_CLOSE :=, INSTANCE := 'AV-24.21', RESTART :=, VISIBILITY :=, OPdwCmd :=, QdwState =>, QwState =>, QCLOSING =>, QCLOSE =>, QOPENING =>, QOPEN =>, QCMD_OP => "AV-24.21", QMON =>, QMON_ERR =>, QMON_T =>, QMON_T_CLOSE =>, QMAN_AUT =>, QREMOTE =>, QSIM =>, QLOCK =>, QERR =>, QERR_EXT =>, QwAlarm =>)
   END_RUNG
   RUNG wire#powerrail
      Contact( "AV-24.21" )
   END_RUNG wire#w1
   RUNG wire#powerrail
      I_Contact( "AV-24.21" )
   END_RUNG wire#w2
   // the same network as SCL:
   #"AV-24.21"(LOCK := #lock,   // "Valve"
               LIOP_SEL := #Init,
               L_AUT := #Init,
               L_REMOTE := #Init,
               L_RESET := #Reset,
               FB_OPEN := "AV-24.21",
               FB_CLOSE := NOT "AV-24.21",
               L_MON := #Init,
               INSTANCE := 'AV-24.21',
               QCMD_OP => "AV-24.21");
END_REGION

REGION Network 26: AV-24.22
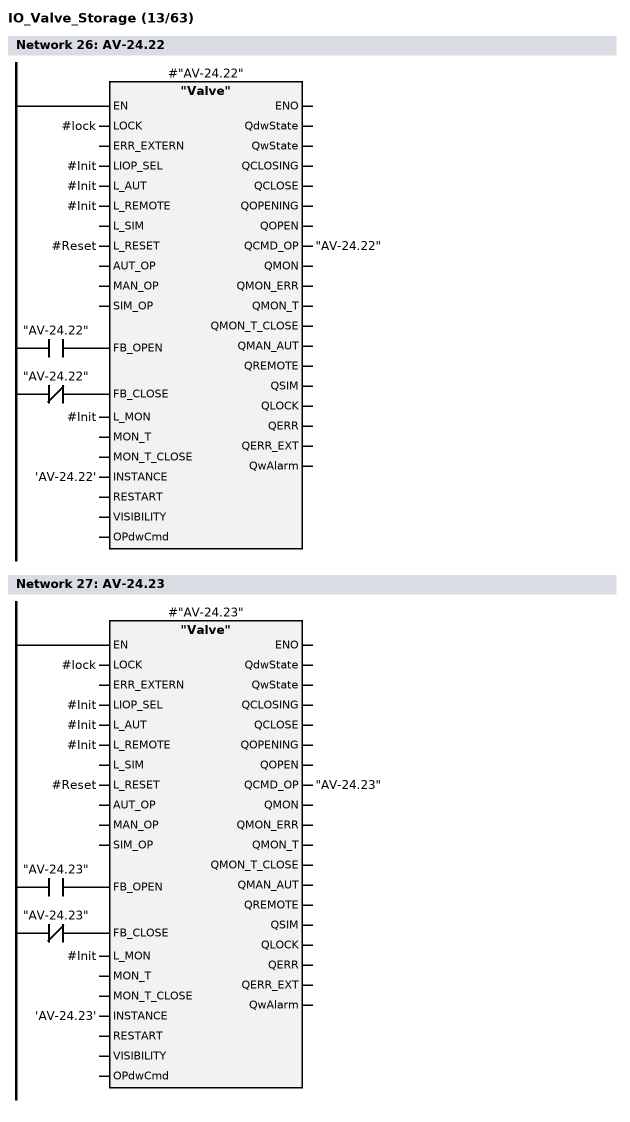
   RUNG wire#powerrail
      #"AV-24.22"(FB_OPEN := wire#w1, FB_CLOSE := wire#w2, LOCK := #lock, ERR_EXTERN :=, LIOP_SEL := #Init, L_AUT := #Init, L_REMOTE := #Init, L_SIM :=, L_RESET := #Reset, AUT_OP :=, MAN_OP :=, SIM_OP :=, L_MON := #Init, MON_T :=, MON_T_CLOSE :=, INSTANCE := 'AV-24.22', RESTART :=, VISIBILITY :=, OPdwCmd :=, QdwState =>, QwState =>, QCLOSING =>, QCLOSE =>, QOPENING =>, QOPEN =>, QCMD_OP => "AV-24.22", QMON =>, QMON_ERR =>, QMON_T =>, QMON_T_CLOSE =>, QMAN_AUT =>, QREMOTE =>, QSIM =>, QLOCK =>, QERR =>, QERR_EXT =>, QwAlarm =>)
   END_RUNG
   RUNG wire#powerrail
      Contact( "AV-24.22" )
   END_RUNG wire#w1
   RUNG wire#powerrail
      I_Contact( "AV-24.22" )
   END_RUNG wire#w2
   // the same network as SCL:
   #"AV-24.22"(LOCK := #lock,   // "Valve"
               LIOP_SEL := #Init,
               L_AUT := #Init,
               L_REMOTE := #Init,
               L_RESET := #Reset,
               FB_OPEN := "AV-24.22",
               FB_CLOSE := NOT "AV-24.22",
               L_MON := #Init,
               INSTANCE := 'AV-24.22',
               QCMD_OP => "AV-24.22");
END_REGION

REGION Network 27: AV-24.23
   RUNG wire#powerrail
      #"AV-24.23"(FB_OPEN := wire#w1, FB_CLOSE := wire#w2, LOCK := #lock, ERR_EXTERN :=, LIOP_SEL := #Init, L_AUT := #Init, L_REMOTE := #Init, L_SIM :=, L_RESET := #Reset, AUT_OP :=, MAN_OP :=, SIM_OP :=, L_MON := #Init, MON_T :=, MON_T_CLOSE :=, INSTANCE := 'AV-24.23', RESTART :=, VISIBILITY :=, OPdwCmd :=, QdwState =>, QwState =>, QCLOSING =>, QCLOSE =>, QOPENING =>, QOPEN =>, QCMD_OP => "AV-24.23", QMON =>, QMON_ERR =>, QMON_T =>, QMON_T_CLOSE =>, QMAN_AUT =>, QREMOTE =>, QSIM =>, QLOCK =>, QERR =>, QERR_EXT =>, QwAlarm =>)
   END_RUNG
   RUNG wire#powerrail
      Contact( "AV-24.23" )
   END_RUNG wire#w1
   RUNG wire#powerrail
      I_Contact( "AV-24.23" )
   END_RUNG wire#w2
   // the same network as SCL:
   #"AV-24.23"(LOCK := #lock,   // "Valve"
               LIOP_SEL := #Init,
               L_AUT := #Init,
               L_REMOTE := #Init,
               L_RESET := #Reset,
               FB_OPEN := "AV-24.23",
               FB_CLOSE := NOT "AV-24.23",
               L_MON := #Init,
               INSTANCE := 'AV-24.23',
               QCMD_OP => "AV-24.23");
END_REGION

REGION Network 28: AV-24.24
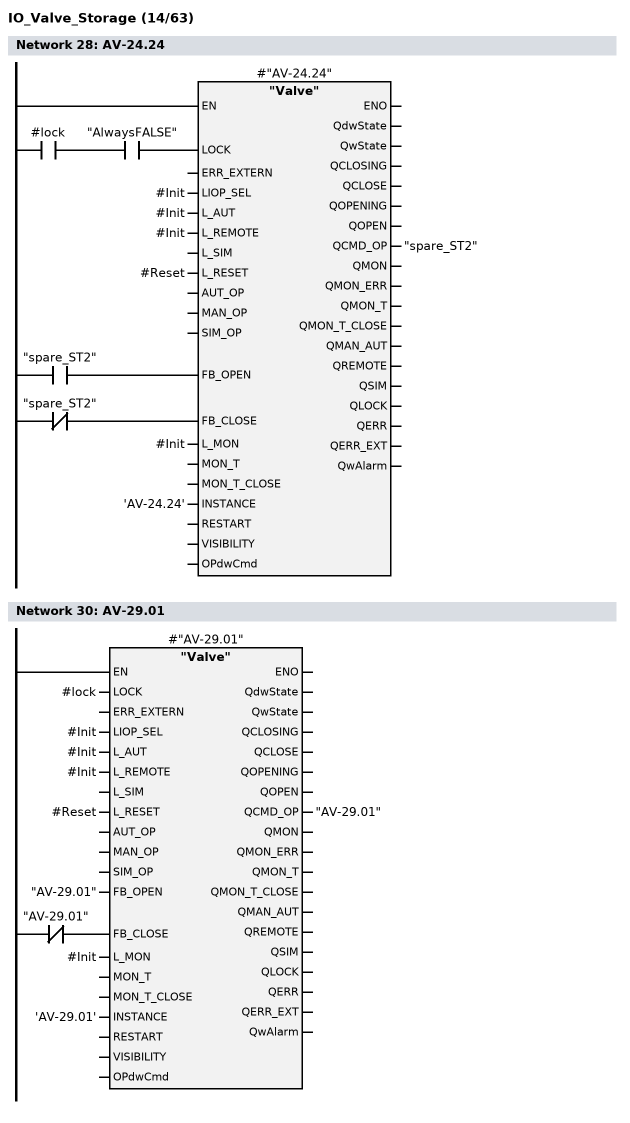
   RUNG wire#powerrail
      #"AV-24.24"(LOCK := wire#w1, FB_OPEN := wire#w2, FB_CLOSE := wire#w3, ERR_EXTERN :=, LIOP_SEL := #Init, L_AUT := #Init, L_REMOTE := #Init, L_SIM :=, L_RESET := #Reset, AUT_OP :=, MAN_OP :=, SIM_OP :=, L_MON := #Init, MON_T :=, MON_T_CLOSE :=, INSTANCE := 'AV-24.24', RESTART :=, VISIBILITY :=, OPdwCmd :=, QdwState =>, QwState =>, QCLOSING =>, QCLOSE =>, QOPENING =>, QOPEN =>, QCMD_OP => "spare_ST2", QMON =>, QMON_ERR =>, QMON_T =>, QMON_T_CLOSE =>, QMAN_AUT =>, QREMOTE =>, QSIM =>, QLOCK =>, QERR =>, QERR_EXT =>, QwAlarm =>)
   END_RUNG
   RUNG wire#powerrail
      Contact( #lock )
      Contact( "AlwaysFALSE" )
   END_RUNG wire#w1
   RUNG wire#powerrail
      Contact( "spare_ST2" )
   END_RUNG wire#w2
   RUNG wire#powerrail
      I_Contact( "spare_ST2" )
   END_RUNG wire#w3
   // the same network as SCL:
   #"AV-24.24"(LOCK := #lock AND "AlwaysFALSE",   // "Valve"
               LIOP_SEL := #Init,
               L_AUT := #Init,
               L_REMOTE := #Init,
               L_RESET := #Reset,
               FB_OPEN := "spare_ST2",
               FB_CLOSE := NOT "spare_ST2",
               L_MON := #Init,
               INSTANCE := 'AV-24.24',
               QCMD_OP => "spare_ST2");
END_REGION

REGION Network 30: AV-29.01
   RUNG wire#powerrail
      #"AV-29.01"(FB_CLOSE := wire#w1, LOCK := #lock, ERR_EXTERN :=, LIOP_SEL := #Init, L_AUT := #Init, L_REMOTE := #Init, L_SIM :=, L_RESET := #Reset, AUT_OP :=, MAN_OP :=, SIM_OP :=, FB_OPEN := "AV-29.01", L_MON := #Init, MON_T :=, MON_T_CLOSE :=, INSTANCE := 'AV-29.01', RESTART :=, VISIBILITY :=, OPdwCmd :=, QdwState =>, QwState =>, QCLOSING =>, QCLOSE =>, QOPENING =>, QOPEN =>, QCMD_OP => "AV-29.01", QMON =>, QMON_ERR =>, QMON_T =>, QMON_T_CLOSE =>, QMAN_AUT =>, QREMOTE =>, QSIM =>, QLOCK =>, QERR =>, QERR_EXT =>, QwAlarm =>)
   END_RUNG
   RUNG wire#powerrail
      I_Contact( "AV-29.01" )
   END_RUNG wire#w1
   // the same network as SCL:
   #"AV-29.01"(LOCK := #lock,   // "Valve"
               LIOP_SEL := #Init,
               L_AUT := #Init,
               L_REMOTE := #Init,
               L_RESET := #Reset,
               FB_OPEN := "AV-29.01",
               FB_CLOSE := NOT "AV-29.01",
               L_MON := #Init,
               INSTANCE := 'AV-29.01',
               QCMD_OP => "AV-29.01");
END_REGION

REGION Network 31: AV-29.02
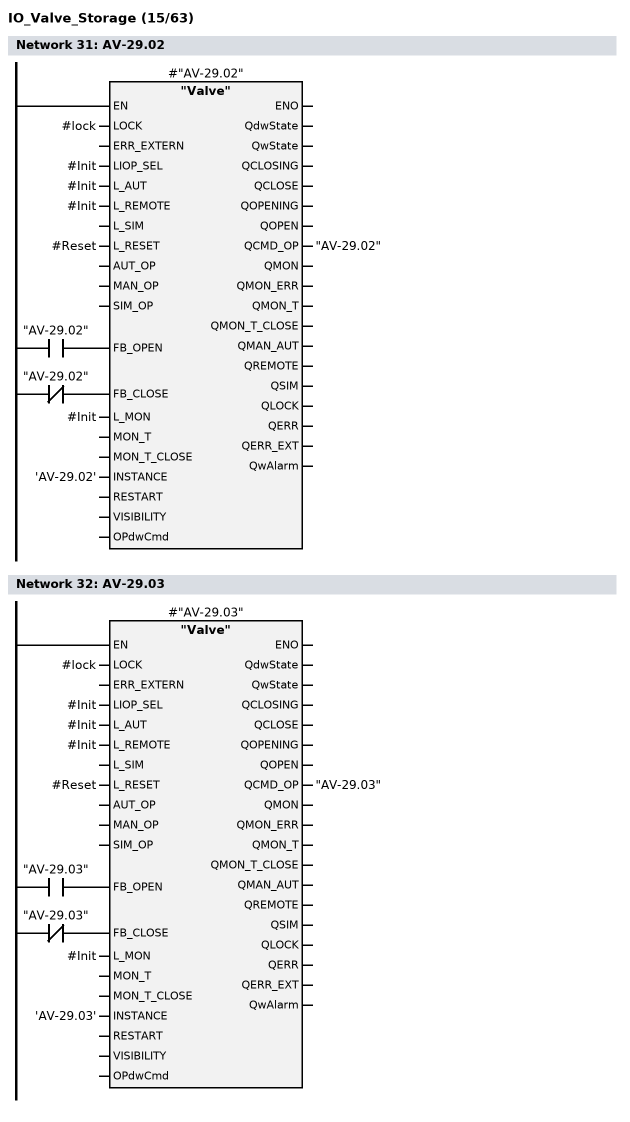
   RUNG wire#powerrail
      #"AV-29.02"(FB_OPEN := wire#w1, FB_CLOSE := wire#w2, LOCK := #lock, ERR_EXTERN :=, LIOP_SEL := #Init, L_AUT := #Init, L_REMOTE := #Init, L_SIM :=, L_RESET := #Reset, AUT_OP :=, MAN_OP :=, SIM_OP :=, L_MON := #Init, MON_T :=, MON_T_CLOSE :=, INSTANCE := 'AV-29.02', RESTART :=, VISIBILITY :=, OPdwCmd :=, QdwState =>, QwState =>, QCLOSING =>, QCLOSE =>, QOPENING =>, QOPEN =>, QCMD_OP => "AV-29.02", QMON =>, QMON_ERR =>, QMON_T =>, QMON_T_CLOSE =>, QMAN_AUT =>, QREMOTE =>, QSIM =>, QLOCK =>, QERR =>, QERR_EXT =>, QwAlarm =>)
   END_RUNG
   RUNG wire#powerrail
      Contact( "AV-29.02" )
   END_RUNG wire#w1
   RUNG wire#powerrail
      I_Contact( "AV-29.02" )
   END_RUNG wire#w2
   // the same network as SCL:
   #"AV-29.02"(LOCK := #lock,   // "Valve"
               LIOP_SEL := #Init,
               L_AUT := #Init,
               L_REMOTE := #Init,
               L_RESET := #Reset,
               FB_OPEN := "AV-29.02",
               FB_CLOSE := NOT "AV-29.02",
               L_MON := #Init,
               INSTANCE := 'AV-29.02',
               QCMD_OP => "AV-29.02");
END_REGION

REGION Network 32: AV-29.03
   RUNG wire#powerrail
      #"AV-29.03"(FB_OPEN := wire#w1, FB_CLOSE := wire#w2, LOCK := #lock, ERR_EXTERN :=, LIOP_SEL := #Init, L_AUT := #Init, L_REMOTE := #Init, L_SIM :=, L_RESET := #Reset, AUT_OP :=, MAN_OP :=, SIM_OP :=, L_MON := #Init, MON_T :=, MON_T_CLOSE :=, INSTANCE := 'AV-29.03', RESTART :=, VISIBILITY :=, OPdwCmd :=, QdwState =>, QwState =>, QCLOSING =>, QCLOSE =>, QOPENING =>, QOPEN =>, QCMD_OP => "AV-29.03", QMON =>, QMON_ERR =>, QMON_T =>, QMON_T_CLOSE =>, QMAN_AUT =>, QREMOTE =>, QSIM =>, QLOCK =>, QERR =>, QERR_EXT =>, QwAlarm =>)
   END_RUNG
   RUNG wire#powerrail
      Contact( "AV-29.03" )
   END_RUNG wire#w1
   RUNG wire#powerrail
      I_Contact( "AV-29.03" )
   END_RUNG wire#w2
   // the same network as SCL:
   #"AV-29.03"(LOCK := #lock,   // "Valve"
               LIOP_SEL := #Init,
               L_AUT := #Init,
               L_REMOTE := #Init,
               L_RESET := #Reset,
               FB_OPEN := "AV-29.03",
               FB_CLOSE := NOT "AV-29.03",
               L_MON := #Init,
               INSTANCE := 'AV-29.03',
               QCMD_OP => "AV-29.03");
END_REGION

REGION Network 33: AV-29.04
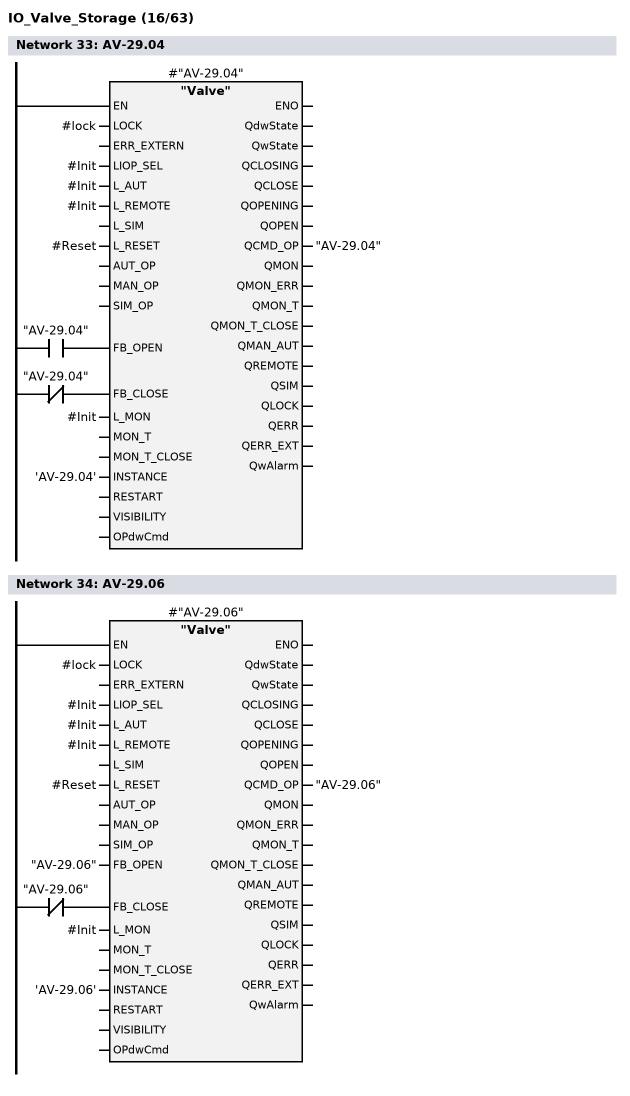
   RUNG wire#powerrail
      #"AV-29.04"(FB_OPEN := wire#w1, FB_CLOSE := wire#w2, LOCK := #lock, ERR_EXTERN :=, LIOP_SEL := #Init, L_AUT := #Init, L_REMOTE := #Init, L_SIM :=, L_RESET := #Reset, AUT_OP :=, MAN_OP :=, SIM_OP :=, L_MON := #Init, MON_T :=, MON_T_CLOSE :=, INSTANCE := 'AV-29.04', RESTART :=, VISIBILITY :=, OPdwCmd :=, QdwState =>, QwState =>, QCLOSING =>, QCLOSE =>, QOPENING =>, QOPEN =>, QCMD_OP => "AV-29.04", QMON =>, QMON_ERR =>, QMON_T =>, QMON_T_CLOSE =>, QMAN_AUT =>, QREMOTE =>, QSIM =>, QLOCK =>, QERR =>, QERR_EXT =>, QwAlarm =>)
   END_RUNG
   RUNG wire#powerrail
      Contact( "AV-29.04" )
   END_RUNG wire#w1
   RUNG wire#powerrail
      I_Contact( "AV-29.04" )
   END_RUNG wire#w2
   // the same network as SCL:
   #"AV-29.04"(LOCK := #lock,   // "Valve"
               LIOP_SEL := #Init,
               L_AUT := #Init,
               L_REMOTE := #Init,
               L_RESET := #Reset,
               FB_OPEN := "AV-29.04",
               FB_CLOSE := NOT "AV-29.04",
               L_MON := #Init,
               INSTANCE := 'AV-29.04',
               QCMD_OP => "AV-29.04");
END_REGION

REGION Network 34: AV-29.06
   RUNG wire#powerrail
      #"AV-29.06"(FB_CLOSE := wire#w1, LOCK := #lock, ERR_EXTERN :=, LIOP_SEL := #Init, L_AUT := #Init, L_REMOTE := #Init, L_SIM :=, L_RESET := #Reset, AUT_OP :=, MAN_OP :=, SIM_OP :=, FB_OPEN := "AV-29.06", L_MON := #Init, MON_T :=, MON_T_CLOSE :=, INSTANCE := 'AV-29.06', RESTART :=, VISIBILITY :=, OPdwCmd :=, QdwState =>, QwState =>, QCLOSING =>, QCLOSE =>, QOPENING =>, QOPEN =>, QCMD_OP => "AV-29.06", QMON =>, QMON_ERR =>, QMON_T =>, QMON_T_CLOSE =>, QMAN_AUT =>, QREMOTE =>, QSIM =>, QLOCK =>, QERR =>, QERR_EXT =>, QwAlarm =>)
   END_RUNG
   RUNG wire#powerrail
      I_Contact( "AV-29.06" )
   END_RUNG wire#w1
   // the same network as SCL:
   #"AV-29.06"(LOCK := #lock,   // "Valve"
               LIOP_SEL := #Init,
               L_AUT := #Init,
               L_REMOTE := #Init,
               L_RESET := #Reset,
               FB_OPEN := "AV-29.06",
               FB_CLOSE := NOT "AV-29.06",
               L_MON := #Init,
               INSTANCE := 'AV-29.06',
               QCMD_OP => "AV-29.06");
END_REGION

REGION Network 36: AV-33.01
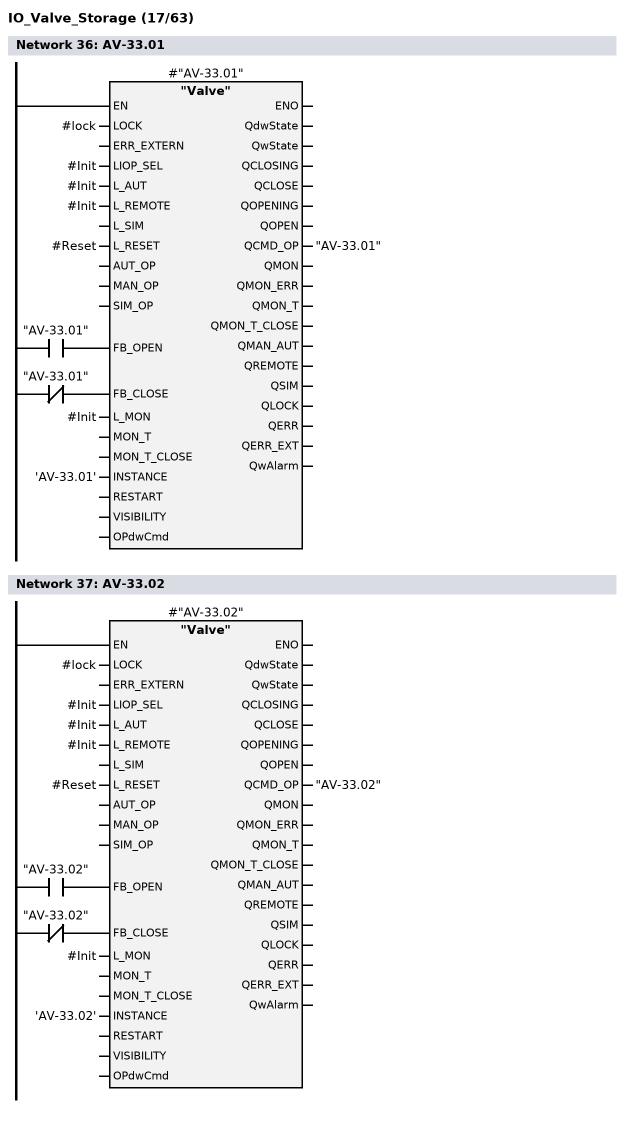
   RUNG wire#powerrail
      #"AV-33.01"(FB_OPEN := wire#w1, FB_CLOSE := wire#w2, LOCK := #lock, ERR_EXTERN :=, LIOP_SEL := #Init, L_AUT := #Init, L_REMOTE := #Init, L_SIM :=, L_RESET := #Reset, AUT_OP :=, MAN_OP :=, SIM_OP :=, L_MON := #Init, MON_T :=, MON_T_CLOSE :=, INSTANCE := 'AV-33.01', RESTART :=, VISIBILITY :=, OPdwCmd :=, QdwState =>, QwState =>, QCLOSING =>, QCLOSE =>, QOPENING =>, QOPEN =>, QCMD_OP => "AV-33.01", QMON =>, QMON_ERR =>, QMON_T =>, QMON_T_CLOSE =>, QMAN_AUT =>, QREMOTE =>, QSIM =>, QLOCK =>, QERR =>, QERR_EXT =>, QwAlarm =>)
   END_RUNG
   RUNG wire#powerrail
      Contact( "AV-33.01" )
   END_RUNG wire#w1
   RUNG wire#powerrail
      I_Contact( "AV-33.01" )
   END_RUNG wire#w2
   // the same network as SCL:
   #"AV-33.01"(LOCK := #lock,   // "Valve"
               LIOP_SEL := #Init,
               L_AUT := #Init,
               L_REMOTE := #Init,
               L_RESET := #Reset,
               FB_OPEN := "AV-33.01",
               FB_CLOSE := NOT "AV-33.01",
               L_MON := #Init,
               INSTANCE := 'AV-33.01',
               QCMD_OP => "AV-33.01");
END_REGION

REGION Network 37: AV-33.02
   RUNG wire#powerrail
      #"AV-33.02"(FB_OPEN := wire#w1, FB_CLOSE := wire#w2, LOCK := #lock, ERR_EXTERN :=, LIOP_SEL := #Init, L_AUT := #Init, L_REMOTE := #Init, L_SIM :=, L_RESET := #Reset, AUT_OP :=, MAN_OP :=, SIM_OP :=, L_MON := #Init, MON_T :=, MON_T_CLOSE :=, INSTANCE := 'AV-33.02', RESTART :=, VISIBILITY :=, OPdwCmd :=, QdwState =>, QwState =>, QCLOSING =>, QCLOSE =>, QOPENING =>, QOPEN =>, QCMD_OP => "AV-33.02", QMON =>, QMON_ERR =>, QMON_T =>, QMON_T_CLOSE =>, QMAN_AUT =>, QREMOTE =>, QSIM =>, QLOCK =>, QERR =>, QERR_EXT =>, QwAlarm =>)
   END_RUNG
   RUNG wire#powerrail
      Contact( "AV-33.02" )
   END_RUNG wire#w1
   RUNG wire#powerrail
      I_Contact( "AV-33.02" )
   END_RUNG wire#w2
   // the same network as SCL:
   #"AV-33.02"(LOCK := #lock,   // "Valve"
               LIOP_SEL := #Init,
               L_AUT := #Init,
               L_REMOTE := #Init,
               L_RESET := #Reset,
               FB_OPEN := "AV-33.02",
               FB_CLOSE := NOT "AV-33.02",
               L_MON := #Init,
               INSTANCE := 'AV-33.02',
               QCMD_OP => "AV-33.02");
END_REGION

REGION Network 38: AV-33.03
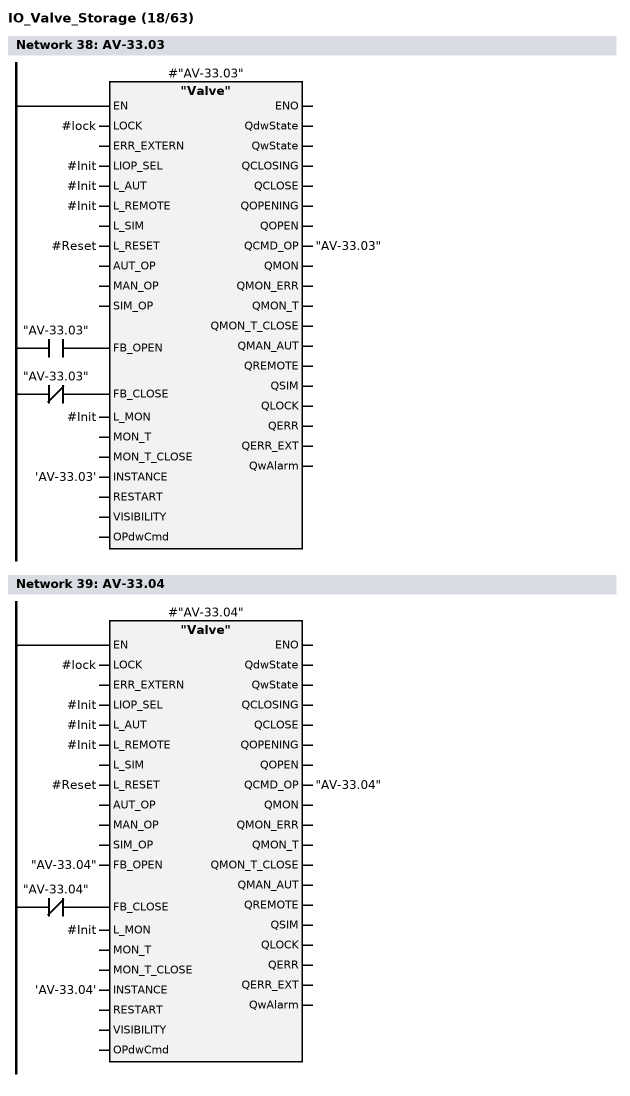
   RUNG wire#powerrail
      #"AV-33.03"(FB_OPEN := wire#w1, FB_CLOSE := wire#w2, LOCK := #lock, ERR_EXTERN :=, LIOP_SEL := #Init, L_AUT := #Init, L_REMOTE := #Init, L_SIM :=, L_RESET := #Reset, AUT_OP :=, MAN_OP :=, SIM_OP :=, L_MON := #Init, MON_T :=, MON_T_CLOSE :=, INSTANCE := 'AV-33.03', RESTART :=, VISIBILITY :=, OPdwCmd :=, QdwState =>, QwState =>, QCLOSING =>, QCLOSE =>, QOPENING =>, QOPEN =>, QCMD_OP => "AV-33.03", QMON =>, QMON_ERR =>, QMON_T =>, QMON_T_CLOSE =>, QMAN_AUT =>, QREMOTE =>, QSIM =>, QLOCK =>, QERR =>, QERR_EXT =>, QwAlarm =>)
   END_RUNG
   RUNG wire#powerrail
      Contact( "AV-33.03" )
   END_RUNG wire#w1
   RUNG wire#powerrail
      I_Contact( "AV-33.03" )
   END_RUNG wire#w2
   // the same network as SCL:
   #"AV-33.03"(LOCK := #lock,   // "Valve"
               LIOP_SEL := #Init,
               L_AUT := #Init,
               L_REMOTE := #Init,
               L_RESET := #Reset,
               FB_OPEN := "AV-33.03",
               FB_CLOSE := NOT "AV-33.03",
               L_MON := #Init,
               INSTANCE := 'AV-33.03',
               QCMD_OP => "AV-33.03");
END_REGION

REGION Network 39: AV-33.04
   RUNG wire#powerrail
      #"AV-33.04"(FB_CLOSE := wire#w1, LOCK := #lock, ERR_EXTERN :=, LIOP_SEL := #Init, L_AUT := #Init, L_REMOTE := #Init, L_SIM :=, L_RESET := #Reset, AUT_OP :=, MAN_OP :=, SIM_OP :=, FB_OPEN := "AV-33.04", L_MON := #Init, MON_T :=, MON_T_CLOSE :=, INSTANCE := 'AV-33.04', RESTART :=, VISIBILITY :=, OPdwCmd :=, QdwState =>, QwState =>, QCLOSING =>, QCLOSE =>, QOPENING =>, QOPEN =>, QCMD_OP => "AV-33.04", QMON =>, QMON_ERR =>, QMON_T =>, QMON_T_CLOSE =>, QMAN_AUT =>, QREMOTE =>, QSIM =>, QLOCK =>, QERR =>, QERR_EXT =>, QwAlarm =>)
   END_RUNG
   RUNG wire#powerrail
      I_Contact( "AV-33.04" )
   END_RUNG wire#w1
   // the same network as SCL:
   #"AV-33.04"(LOCK := #lock,   // "Valve"
               LIOP_SEL := #Init,
               L_AUT := #Init,
               L_REMOTE := #Init,
               L_RESET := #Reset,
               FB_OPEN := "AV-33.04",
               FB_CLOSE := NOT "AV-33.04",
               L_MON := #Init,
               INSTANCE := 'AV-33.04',
               QCMD_OP => "AV-33.04");
END_REGION

REGION Network 40: AV-33.05
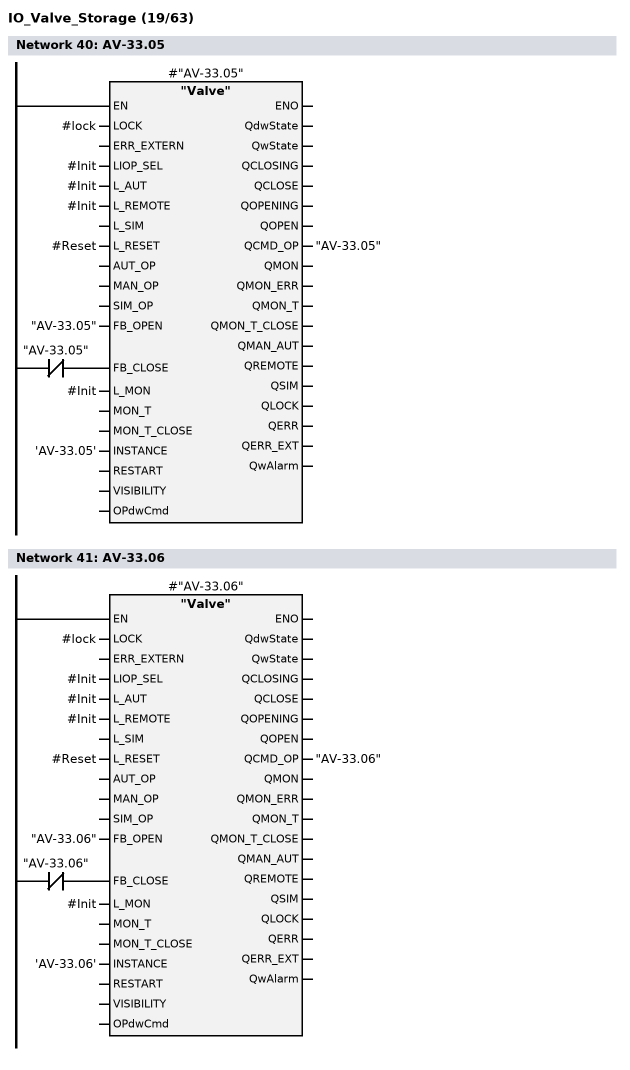
   RUNG wire#powerrail
      #"AV-33.05"(FB_CLOSE := wire#w1, LOCK := #lock, ERR_EXTERN :=, LIOP_SEL := #Init, L_AUT := #Init, L_REMOTE := #Init, L_SIM :=, L_RESET := #Reset, AUT_OP :=, MAN_OP :=, SIM_OP :=, FB_OPEN := "AV-33.05", L_MON := #Init, MON_T :=, MON_T_CLOSE :=, INSTANCE := 'AV-33.05', RESTART :=, VISIBILITY :=, OPdwCmd :=, QdwState =>, QwState =>, QCLOSING =>, QCLOSE =>, QOPENING =>, QOPEN =>, QCMD_OP => "AV-33.05", QMON =>, QMON_ERR =>, QMON_T =>, QMON_T_CLOSE =>, QMAN_AUT =>, QREMOTE =>, QSIM =>, QLOCK =>, QERR =>, QERR_EXT =>, QwAlarm =>)
   END_RUNG
   RUNG wire#powerrail
      I_Contact( "AV-33.05" )
   END_RUNG wire#w1
   // the same network as SCL:
   #"AV-33.05"(LOCK := #lock,   // "Valve"
               LIOP_SEL := #Init,
               L_AUT := #Init,
               L_REMOTE := #Init,
               L_RESET := #Reset,
               FB_OPEN := "AV-33.05",
               FB_CLOSE := NOT "AV-33.05",
               L_MON := #Init,
               INSTANCE := 'AV-33.05',
               QCMD_OP => "AV-33.05");
END_REGION

REGION Network 41: AV-33.06
   RUNG wire#powerrail
      #"AV-33.06"(FB_CLOSE := wire#w1, LOCK := #lock, ERR_EXTERN :=, LIOP_SEL := #Init, L_AUT := #Init, L_REMOTE := #Init, L_SIM :=, L_RESET := #Reset, AUT_OP :=, MAN_OP :=, SIM_OP :=, FB_OPEN := "AV-33.06", L_MON := #Init, MON_T :=, MON_T_CLOSE :=, INSTANCE := 'AV-33.06', RESTART :=, VISIBILITY :=, OPdwCmd :=, QdwState =>, QwState =>, QCLOSING =>, QCLOSE =>, QOPENING =>, QOPEN =>, QCMD_OP => "AV-33.06", QMON =>, QMON_ERR =>, QMON_T =>, QMON_T_CLOSE =>, QMAN_AUT =>, QREMOTE =>, QSIM =>, QLOCK =>, QERR =>, QERR_EXT =>, QwAlarm =>)
   END_RUNG
   RUNG wire#powerrail
      I_Contact( "AV-33.06" )
   END_RUNG wire#w1
   // the same network as SCL:
   #"AV-33.06"(LOCK := #lock,   // "Valve"
               LIOP_SEL := #Init,
               L_AUT := #Init,
               L_REMOTE := #Init,
               L_RESET := #Reset,
               FB_OPEN := "AV-33.06",
               FB_CLOSE := NOT "AV-33.06",
               L_MON := #Init,
               INSTANCE := 'AV-33.06',
               QCMD_OP => "AV-33.06");
END_REGION

REGION Network 42: AV-33.07
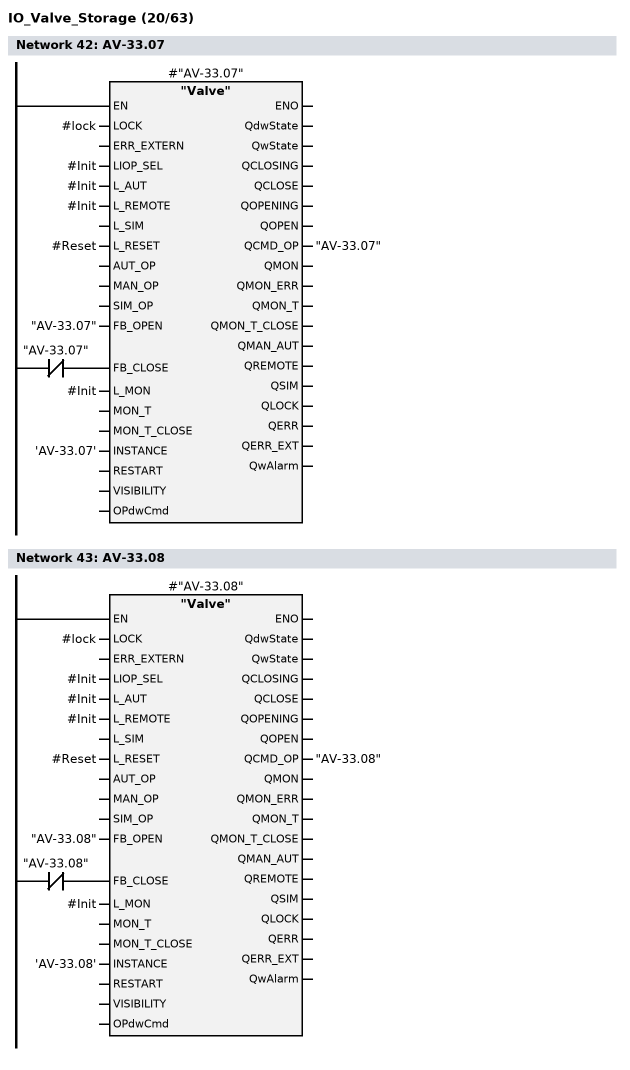
   RUNG wire#powerrail
      #"AV-33.07"(FB_CLOSE := wire#w1, LOCK := #lock, ERR_EXTERN :=, LIOP_SEL := #Init, L_AUT := #Init, L_REMOTE := #Init, L_SIM :=, L_RESET := #Reset, AUT_OP :=, MAN_OP :=, SIM_OP :=, FB_OPEN := "AV-33.07", L_MON := #Init, MON_T :=, MON_T_CLOSE :=, INSTANCE := 'AV-33.07', RESTART :=, VISIBILITY :=, OPdwCmd :=, QdwState =>, QwState =>, QCLOSING =>, QCLOSE =>, QOPENING =>, QOPEN =>, QCMD_OP => "AV-33.07", QMON =>, QMON_ERR =>, QMON_T =>, QMON_T_CLOSE =>, QMAN_AUT =>, QREMOTE =>, QSIM =>, QLOCK =>, QERR =>, QERR_EXT =>, QwAlarm =>)
   END_RUNG
   RUNG wire#powerrail
      I_Contact( "AV-33.07" )
   END_RUNG wire#w1
   // the same network as SCL:
   #"AV-33.07"(LOCK := #lock,   // "Valve"
               LIOP_SEL := #Init,
               L_AUT := #Init,
               L_REMOTE := #Init,
               L_RESET := #Reset,
               FB_OPEN := "AV-33.07",
               FB_CLOSE := NOT "AV-33.07",
               L_MON := #Init,
               INSTANCE := 'AV-33.07',
               QCMD_OP => "AV-33.07");
END_REGION

REGION Network 43: AV-33.08
   RUNG wire#powerrail
      #"AV-33.08"(FB_CLOSE := wire#w1, LOCK := #lock, ERR_EXTERN :=, LIOP_SEL := #Init, L_AUT := #Init, L_REMOTE := #Init, L_SIM :=, L_RESET := #Reset, AUT_OP :=, MAN_OP :=, SIM_OP :=, FB_OPEN := "AV-33.08", L_MON := #Init, MON_T :=, MON_T_CLOSE :=, INSTANCE := 'AV-33.08', RESTART :=, VISIBILITY :=, OPdwCmd :=, QdwState =>, QwState =>, QCLOSING =>, QCLOSE =>, QOPENING =>, QOPEN =>, QCMD_OP => "AV-33.08", QMON =>, QMON_ERR =>, QMON_T =>, QMON_T_CLOSE =>, QMAN_AUT =>, QREMOTE =>, QSIM =>, QLOCK =>, QERR =>, QERR_EXT =>, QwAlarm =>)
   END_RUNG
   RUNG wire#powerrail
      I_Contact( "AV-33.08" )
   END_RUNG wire#w1
   // the same network as SCL:
   #"AV-33.08"(LOCK := #lock,   // "Valve"
               LIOP_SEL := #Init,
               L_AUT := #Init,
               L_REMOTE := #Init,
               L_RESET := #Reset,
               FB_OPEN := "AV-33.08",
               FB_CLOSE := NOT "AV-33.08",
               L_MON := #Init,
               INSTANCE := 'AV-33.08',
               QCMD_OP => "AV-33.08");
END_REGION

REGION Network 44: AV-33.09
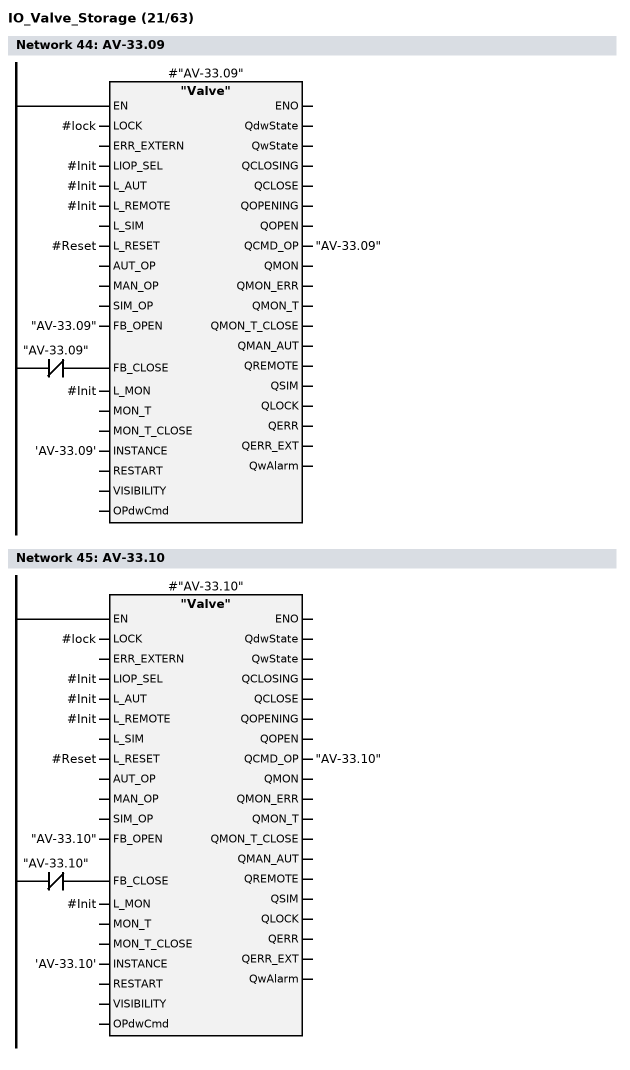
   RUNG wire#powerrail
      #"AV-33.09"(FB_CLOSE := wire#w1, LOCK := #lock, ERR_EXTERN :=, LIOP_SEL := #Init, L_AUT := #Init, L_REMOTE := #Init, L_SIM :=, L_RESET := #Reset, AUT_OP :=, MAN_OP :=, SIM_OP :=, FB_OPEN := "AV-33.09", L_MON := #Init, MON_T :=, MON_T_CLOSE :=, INSTANCE := 'AV-33.09', RESTART :=, VISIBILITY :=, OPdwCmd :=, QdwState =>, QwState =>, QCLOSING =>, QCLOSE =>, QOPENING =>, QOPEN =>, QCMD_OP => "AV-33.09", QMON =>, QMON_ERR =>, QMON_T =>, QMON_T_CLOSE =>, QMAN_AUT =>, QREMOTE =>, QSIM =>, QLOCK =>, QERR =>, QERR_EXT =>, QwAlarm =>)
   END_RUNG
   RUNG wire#powerrail
      I_Contact( "AV-33.09" )
   END_RUNG wire#w1
   // the same network as SCL:
   #"AV-33.09"(LOCK := #lock,   // "Valve"
               LIOP_SEL := #Init,
               L_AUT := #Init,
               L_REMOTE := #Init,
               L_RESET := #Reset,
               FB_OPEN := "AV-33.09",
               FB_CLOSE := NOT "AV-33.09",
               L_MON := #Init,
               INSTANCE := 'AV-33.09',
               QCMD_OP => "AV-33.09");
END_REGION

REGION Network 45: AV-33.10
   RUNG wire#powerrail
      #"AV-33.10"(FB_CLOSE := wire#w1, LOCK := #lock, ERR_EXTERN :=, LIOP_SEL := #Init, L_AUT := #Init, L_REMOTE := #Init, L_SIM :=, L_RESET := #Reset, AUT_OP :=, MAN_OP :=, SIM_OP :=, FB_OPEN := "AV-33.10", L_MON := #Init, MON_T :=, MON_T_CLOSE :=, INSTANCE := 'AV-33.10', RESTART :=, VISIBILITY :=, OPdwCmd :=, QdwState =>, QwState =>, QCLOSING =>, QCLOSE =>, QOPENING =>, QOPEN =>, QCMD_OP => "AV-33.10", QMON =>, QMON_ERR =>, QMON_T =>, QMON_T_CLOSE =>, QMAN_AUT =>, QREMOTE =>, QSIM =>, QLOCK =>, QERR =>, QERR_EXT =>, QwAlarm =>)
   END_RUNG
   RUNG wire#powerrail
      I_Contact( "AV-33.10" )
   END_RUNG wire#w1
   // the same network as SCL:
   #"AV-33.10"(LOCK := #lock,   // "Valve"
               LIOP_SEL := #Init,
               L_AUT := #Init,
               L_REMOTE := #Init,
               L_RESET := #Reset,
               FB_OPEN := "AV-33.10",
               FB_CLOSE := NOT "AV-33.10",
               L_MON := #Init,
               INSTANCE := 'AV-33.10',
               QCMD_OP => "AV-33.10");
END_REGION

REGION Network 46: AV-33.11
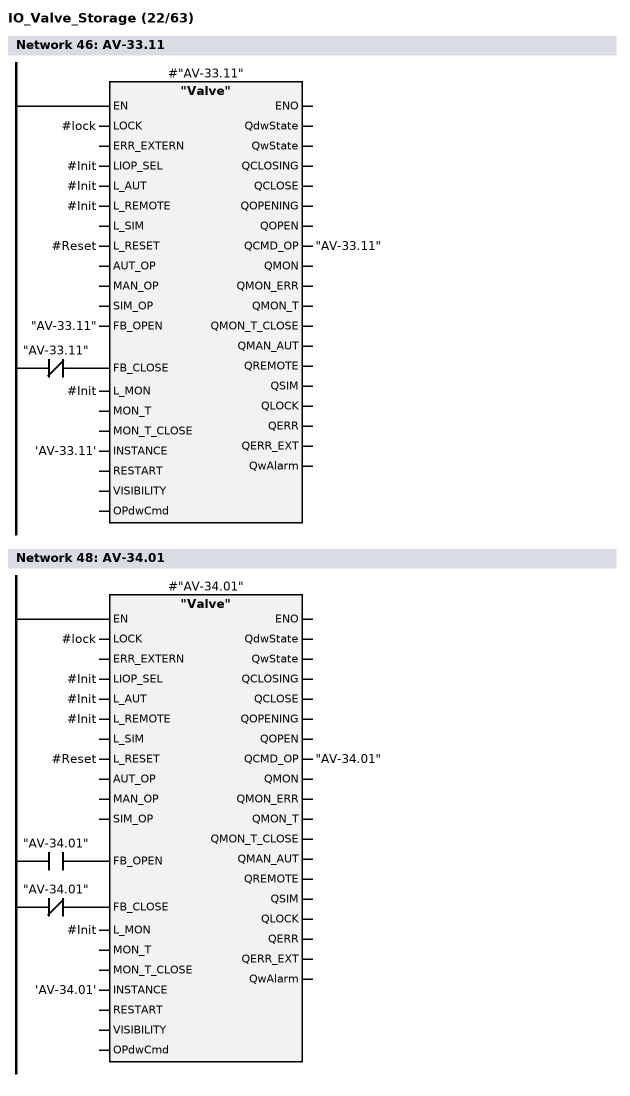
   RUNG wire#powerrail
      #"AV-33.11"(FB_CLOSE := wire#w1, LOCK := #lock, ERR_EXTERN :=, LIOP_SEL := #Init, L_AUT := #Init, L_REMOTE := #Init, L_SIM :=, L_RESET := #Reset, AUT_OP :=, MAN_OP :=, SIM_OP :=, FB_OPEN := "AV-33.11", L_MON := #Init, MON_T :=, MON_T_CLOSE :=, INSTANCE := 'AV-33.11', RESTART :=, VISIBILITY :=, OPdwCmd :=, QdwState =>, QwState =>, QCLOSING =>, QCLOSE =>, QOPENING =>, QOPEN =>, QCMD_OP => "AV-33.11", QMON =>, QMON_ERR =>, QMON_T =>, QMON_T_CLOSE =>, QMAN_AUT =>, QREMOTE =>, QSIM =>, QLOCK =>, QERR =>, QERR_EXT =>, QwAlarm =>)
   END_RUNG
   RUNG wire#powerrail
      I_Contact( "AV-33.11" )
   END_RUNG wire#w1
   // the same network as SCL:
   #"AV-33.11"(LOCK := #lock,   // "Valve"
               LIOP_SEL := #Init,
               L_AUT := #Init,
               L_REMOTE := #Init,
               L_RESET := #Reset,
               FB_OPEN := "AV-33.11",
               FB_CLOSE := NOT "AV-33.11",
               L_MON := #Init,
               INSTANCE := 'AV-33.11',
               QCMD_OP => "AV-33.11");
END_REGION

REGION Network 48: AV-34.01
   RUNG wire#powerrail
      #"AV-34.01"(FB_OPEN := wire#w1, FB_CLOSE := wire#w2, LOCK := #lock, ERR_EXTERN :=, LIOP_SEL := #Init, L_AUT := #Init, L_REMOTE := #Init, L_SIM :=, L_RESET := #Reset, AUT_OP :=, MAN_OP :=, SIM_OP :=, L_MON := #Init, MON_T :=, MON_T_CLOSE :=, INSTANCE := 'AV-34.01', RESTART :=, VISIBILITY :=, OPdwCmd :=, QdwState =>, QwState =>, QCLOSING =>, QCLOSE =>, QOPENING =>, QOPEN =>, QCMD_OP => "AV-34.01", QMON =>, QMON_ERR =>, QMON_T =>, QMON_T_CLOSE =>, QMAN_AUT =>, QREMOTE =>, QSIM =>, QLOCK =>, QERR =>, QERR_EXT =>, QwAlarm =>)
   END_RUNG
   RUNG wire#powerrail
      Contact( "AV-34.01" )
   END_RUNG wire#w1
   RUNG wire#powerrail
      I_Contact( "AV-34.01" )
   END_RUNG wire#w2
   // the same network as SCL:
   #"AV-34.01"(LOCK := #lock,   // "Valve"
               LIOP_SEL := #Init,
               L_AUT := #Init,
               L_REMOTE := #Init,
               L_RESET := #Reset,
               FB_OPEN := "AV-34.01",
               FB_CLOSE := NOT "AV-34.01",
               L_MON := #Init,
               INSTANCE := 'AV-34.01',
               QCMD_OP => "AV-34.01");
END_REGION

REGION Network 49: AV-34.02
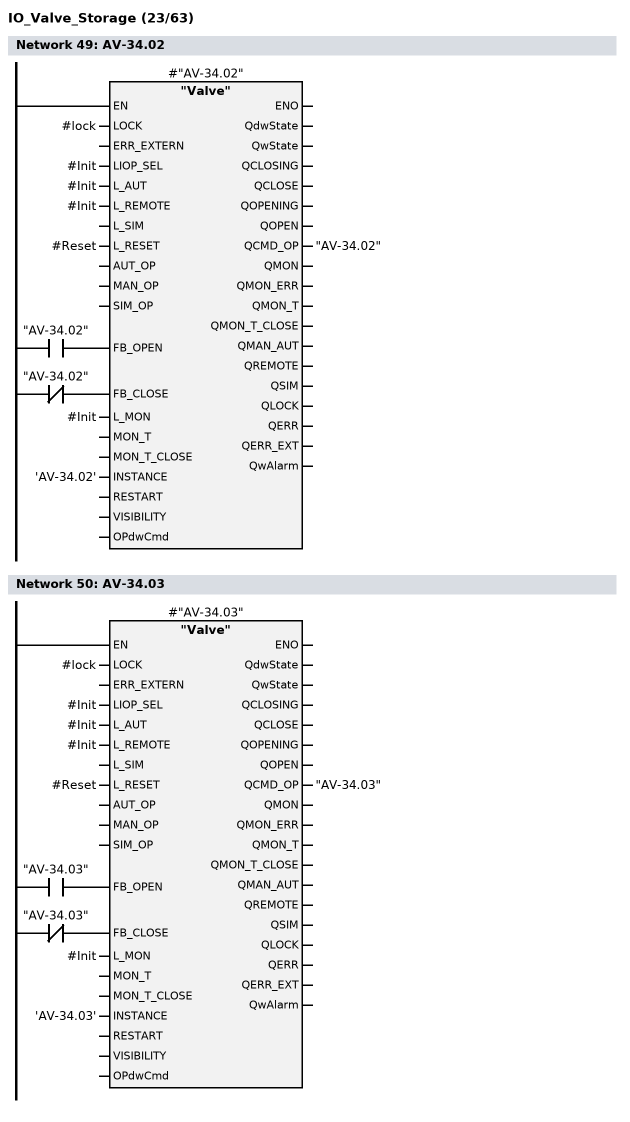
   RUNG wire#powerrail
      #"AV-34.02"(FB_OPEN := wire#w1, FB_CLOSE := wire#w2, LOCK := #lock, ERR_EXTERN :=, LIOP_SEL := #Init, L_AUT := #Init, L_REMOTE := #Init, L_SIM :=, L_RESET := #Reset, AUT_OP :=, MAN_OP :=, SIM_OP :=, L_MON := #Init, MON_T :=, MON_T_CLOSE :=, INSTANCE := 'AV-34.02', RESTART :=, VISIBILITY :=, OPdwCmd :=, QdwState =>, QwState =>, QCLOSING =>, QCLOSE =>, QOPENING =>, QOPEN =>, QCMD_OP => "AV-34.02", QMON =>, QMON_ERR =>, QMON_T =>, QMON_T_CLOSE =>, QMAN_AUT =>, QREMOTE =>, QSIM =>, QLOCK =>, QERR =>, QERR_EXT =>, QwAlarm =>)
   END_RUNG
   RUNG wire#powerrail
      Contact( "AV-34.02" )
   END_RUNG wire#w1
   RUNG wire#powerrail
      I_Contact( "AV-34.02" )
   END_RUNG wire#w2
   // the same network as SCL:
   #"AV-34.02"(LOCK := #lock,   // "Valve"
               LIOP_SEL := #Init,
               L_AUT := #Init,
               L_REMOTE := #Init,
               L_RESET := #Reset,
               FB_OPEN := "AV-34.02",
               FB_CLOSE := NOT "AV-34.02",
               L_MON := #Init,
               INSTANCE := 'AV-34.02',
               QCMD_OP => "AV-34.02");
END_REGION

REGION Network 50: AV-34.03
   RUNG wire#powerrail
      #"AV-34.03"(FB_OPEN := wire#w1, FB_CLOSE := wire#w2, LOCK := #lock, ERR_EXTERN :=, LIOP_SEL := #Init, L_AUT := #Init, L_REMOTE := #Init, L_SIM :=, L_RESET := #Reset, AUT_OP :=, MAN_OP :=, SIM_OP :=, L_MON := #Init, MON_T :=, MON_T_CLOSE :=, INSTANCE := 'AV-34.03', RESTART :=, VISIBILITY :=, OPdwCmd :=, QdwState =>, QwState =>, QCLOSING =>, QCLOSE =>, QOPENING =>, QOPEN =>, QCMD_OP => "AV-34.03", QMON =>, QMON_ERR =>, QMON_T =>, QMON_T_CLOSE =>, QMAN_AUT =>, QREMOTE =>, QSIM =>, QLOCK =>, QERR =>, QERR_EXT =>, QwAlarm =>)
   END_RUNG
   RUNG wire#powerrail
      Contact( "AV-34.03" )
   END_RUNG wire#w1
   RUNG wire#powerrail
      I_Contact( "AV-34.03" )
   END_RUNG wire#w2
   // the same network as SCL:
   #"AV-34.03"(LOCK := #lock,   // "Valve"
               LIOP_SEL := #Init,
               L_AUT := #Init,
               L_REMOTE := #Init,
               L_RESET := #Reset,
               FB_OPEN := "AV-34.03",
               FB_CLOSE := NOT "AV-34.03",
               L_MON := #Init,
               INSTANCE := 'AV-34.03',
               QCMD_OP => "AV-34.03");
END_REGION

REGION Network 51: AV-34.04
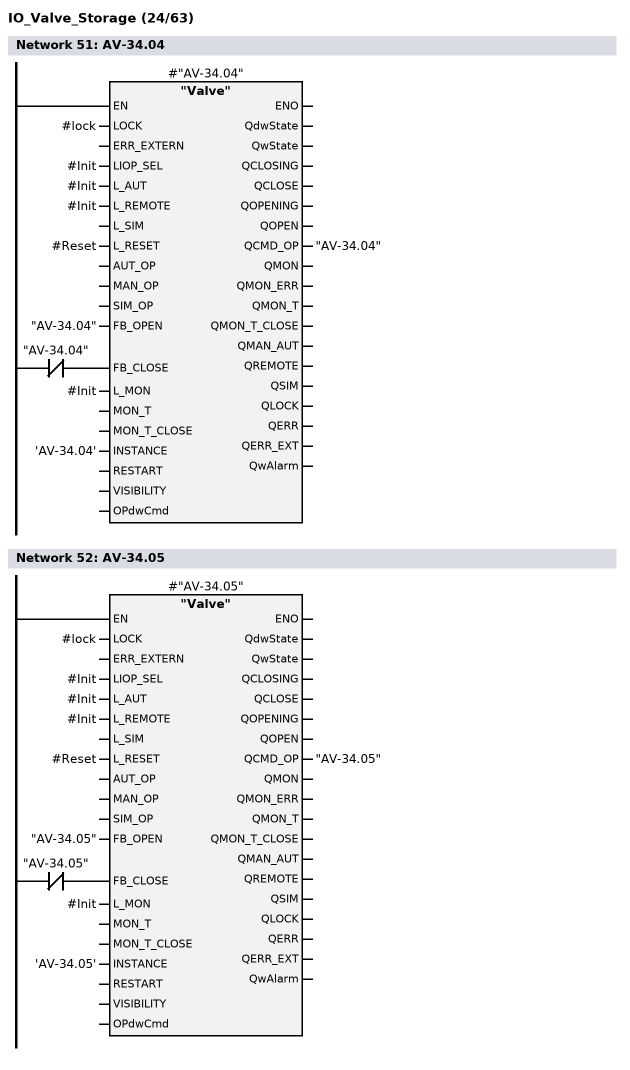
   RUNG wire#powerrail
      #"AV-34.04"(FB_CLOSE := wire#w1, LOCK := #lock, ERR_EXTERN :=, LIOP_SEL := #Init, L_AUT := #Init, L_REMOTE := #Init, L_SIM :=, L_RESET := #Reset, AUT_OP :=, MAN_OP :=, SIM_OP :=, FB_OPEN := "AV-34.04", L_MON := #Init, MON_T :=, MON_T_CLOSE :=, INSTANCE := 'AV-34.04', RESTART :=, VISIBILITY :=, OPdwCmd :=, QdwState =>, QwState =>, QCLOSING =>, QCLOSE =>, QOPENING =>, QOPEN =>, QCMD_OP => "AV-34.04", QMON =>, QMON_ERR =>, QMON_T =>, QMON_T_CLOSE =>, QMAN_AUT =>, QREMOTE =>, QSIM =>, QLOCK =>, QERR =>, QERR_EXT =>, QwAlarm =>)
   END_RUNG
   RUNG wire#powerrail
      I_Contact( "AV-34.04" )
   END_RUNG wire#w1
   // the same network as SCL:
   #"AV-34.04"(LOCK := #lock,   // "Valve"
               LIOP_SEL := #Init,
               L_AUT := #Init,
               L_REMOTE := #Init,
               L_RESET := #Reset,
               FB_OPEN := "AV-34.04",
               FB_CLOSE := NOT "AV-34.04",
               L_MON := #Init,
               INSTANCE := 'AV-34.04',
               QCMD_OP => "AV-34.04");
END_REGION

REGION Network 52: AV-34.05
   RUNG wire#powerrail
      #"AV-34.05"(FB_CLOSE := wire#w1, LOCK := #lock, ERR_EXTERN :=, LIOP_SEL := #Init, L_AUT := #Init, L_REMOTE := #Init, L_SIM :=, L_RESET := #Reset, AUT_OP :=, MAN_OP :=, SIM_OP :=, FB_OPEN := "AV-34.05", L_MON := #Init, MON_T :=, MON_T_CLOSE :=, INSTANCE := 'AV-34.05', RESTART :=, VISIBILITY :=, OPdwCmd :=, QdwState =>, QwState =>, QCLOSING =>, QCLOSE =>, QOPENING =>, QOPEN =>, QCMD_OP => "AV-34.05", QMON =>, QMON_ERR =>, QMON_T =>, QMON_T_CLOSE =>, QMAN_AUT =>, QREMOTE =>, QSIM =>, QLOCK =>, QERR =>, QERR_EXT =>, QwAlarm =>)
   END_RUNG
   RUNG wire#powerrail
      I_Contact( "AV-34.05" )
   END_RUNG wire#w1
   // the same network as SCL:
   #"AV-34.05"(LOCK := #lock,   // "Valve"
               LIOP_SEL := #Init,
               L_AUT := #Init,
               L_REMOTE := #Init,
               L_RESET := #Reset,
               FB_OPEN := "AV-34.05",
               FB_CLOSE := NOT "AV-34.05",
               L_MON := #Init,
               INSTANCE := 'AV-34.05',
               QCMD_OP => "AV-34.05");
END_REGION

REGION Network 53: AV-34.06
